// TwinCAT 3 PLC project WC1
// ProgramVersion: 3.1.4024.0
// libraries:
//   CmpBitmapPool, * (System)
//   Tc2_ModbusSrv, * (Beckhoff Automation GmbH)
//   Tc2_Standard, * (Beckhoff Automation GmbH)
//   Tc2_System, * (Beckhoff Automation GmbH)
//   Tc2_Utilities, * (Beckhoff Automation GmbH)
//   Tc3_Module, * (Beckhoff Automation GmbH)
//   VisuDialogs, * (System)
//   VisuSymbols,3.5.10.0,System
// project tree:
//   DUTs/ SEQ_NAME.TcDUT
//   / GlobalTextList.TcGTLO, PlcTask.TcTTO, Visualization Manager.TcVMO (not stored), VISU_TASK.TcTTO
//   POUs/Auto_Seq/ AUTO_MODE.TcPOU, FB_RunLayerPad.TcPOU, IF_RACK_CHECK.TcPOU, SEQ_A1.TcPOU, SEQ_A2.TcPOU, SEQ_A3.TcPOU, SEQ_A4.TcPOU, SEQ_A5.TcPOU, SEQ_B1.TcPOU, SEQ_B2.TcPOU, SEQ_B3.TcPOU, SEQ_B4.TcPOU, SEQ_B5.TcPOU, SEQ_COSMO.TcPOU, SEQ_CR_PICK.TcPOU, SEQ_CR_PLACE.TcPOU, SEQ_FG.TcPOU, SEQ_FG_A.TcPOU, SEQ_LYR_PD0.TcPOU, SEQ_RW.TcPOU
//   POUs/ COOL_RACK.TcPOU, ESTOP.TcPOU, INFEED_RACK.TcPOU, JIG.TcPOU, LOGGING.TcPOU, MAIN.TcPOU, RESET_SEQ.TcPOU, LOG_TIME_STAMP.TcPOU, SAFETY_SENSOR.TcPOU, TL.TcPOU, TORCHCLEAN.TcPOU, User.TcTLO
//   POUs/GVLs/ GVL.TcGVL, MSG.TcGVL
//   POUs/Kuka IO/ KR1.TcPOU, KR2.TcPOU, KR3.TcPOU, KR4.TcPOU, KR5.TcPOU, KUKA_IO.TcPOU
//   POUs/LOGGING/ FB_UpdateTimeStamp.TcPOU, LOGFILE.TcPOU, LOGPROCESS.TcPOU
//   VISUs/Dialog/ MSG_BOX_RESET.TcVIS, MSG_EOAT.TcVIS, MSG_EOAT_SUCTION.TcVIS, MSG_KR2_BP.TcVIS, MSG_KR4_BP.TcVIS, MSG_KR1_BP.TcVIS, MSG_KR3_BP.TcVIS
//   VISUs/ Footer_Main.TcVIS, Footer_Back.TcVIS, Header.TcVIS, ImagePool.TcIPO (not stored), PAGE_InfeedRack.TcVIS, PAGE_COSMO.TcVIS, PAGE_JIG_C.TcVIS, PAGE_CoolRack.TcVIS, PAGE_JIG_A.TcVIS, PAGE_JIG_B.TcVIS, PAGE_KR1_Tab.TcVIS, PAGE_KR1_Tab_1_100.TcVIS, PAGE_KR1_Tab_1_200.TcVIS, PAGE_MAIN_1.TcVIS, PAGE_TTorch.TcVIS, PAGE_MAIN.TcVIS, PAGE_KR2.TcVIS, PAGE_KR3.TcVIS, PAGE_KR4.TcVIS, PAGE_KR5.TcVIS, PAGE_KR1.TcVIS
// real-time tasks:
//   TASK PlcTask: cycle T#10ms, priority 6, ADS port 350
//   TASK VISU_TASK: cycle T#100000us, priority 8, ADS port 351
// I/O:
//   DEVICE Device 3 (EtherCAT), AmsNetId 169.254.168.184.4.1
//     Term 5 (EK1100) [EK1100 EtherCAT Coupler (2A E-Bus)]
//       Term 12 (EL1889) [EL1889 16Ch. Dig. Input 24V, 3ms, negative]
//       Term 13 (EL1889) [EL1889 16Ch. Dig. Input 24V, 3ms, negative]
//       Term 14 (EL2889) [EL2889 16Ch. Dig. Output 24V, 0.5A, negative]
//       Term 15 (EL9410) [EL9410 E-Bus Power Supplier  (Diagnostics)]
//       Term 16 (EL6695) KR1(KR5) [EL6695 EtherCAT Bridge terminal (Primary)]
//       Term 17 (EL6695) KR2(KR3) [EL6695 EtherCAT Bridge terminal (Primary)]
//       Term 18 (EL6695) KR3(KR2) [EL6695 EtherCAT Bridge terminal (Primary)]
//       Term 19 (EL6695) KR4 [EL6695 EtherCAT Bridge terminal (Primary)]
//       Term 20 (EL6695) KR5(KR1) [EL6695 EtherCAT Bridge terminal (Primary)]
//       Term 21 (EL9011) [EL9011 End Terminal]
// variable links:
//   WC1/WC1 Instance <-> Device 3 (EtherCAT)/Term 5 (EK1100)/Term 12 (EL1889)
//     PlcTask Inputs/GVL.COSMO_NOTOK <-> Channel 12/COSMO NOTOK
//     PlcTask Inputs/GVL.COSMO_OK <-> Channel 11/COSMO OK
//     PlcTask Inputs/GVL.COSMO_Ready <-> Channel 10/COSMO READY
//     PlcTask Inputs/GVL.Conveyor_Full <-> Channel 14/CONVY FULL
//     PlcTask Inputs/GVL.JIGA_Ready <-> Channel 3/JIG A READY
//     PlcTask Inputs/GVL.JIGA_Standby <-> Channel 2/JIG A STANDBY
//     PlcTask Inputs/GVL.JIGB_Ready <-> Channel 5/JIG B READY
//     PlcTask Inputs/GVL.JIGB_Standby <-> Channel 4/JIG B STANDBY
//     PlcTask Inputs/GVL.JIGC_Ready <-> Channel 7/JIG C READY
//     PlcTask Inputs/GVL.JIGC_Standby <-> Channel 6/JIG C STANDBY
//     PlcTask Inputs/GVL.Rework_Empty <-> Channel 15/REWORK EMPTY
//     PlcTask Inputs/GVL.TTorch_Complete <-> Channel 9/TT COMPLETE
//     PlcTask Inputs/GVL.TTorch_Standy <-> Channel 8/TT STANDBY
//     PlcTask Inputs/GVL.VibBowl_Ready <-> Channel 13/VB READY
//     PlcTask Inputs/MAIN.btnEstop <-> Channel 1/Estop
//   WC1/WC1 Instance <-> Device 3 (EtherCAT)/Term 5 (EK1100)/Term 13 (EL1889)
//     PlcTask Inputs/GVL.JIGA_Complete <-> Channel 9/JIGA_Complete
//     PlcTask Inputs/GVL.JIGB_Complete <-> Channel 10/JIGB_Complete
//     PlcTask Inputs/GVL.JIGC_Complete <-> Channel 11/JIGC_Complete
//     PlcTask Inputs/MAIN.btnReset <-> Channel 3/RESET BTN
//     PlcTask Inputs/MAIN.btnStart <-> Channel 1/START BTN
//     PlcTask Inputs/MAIN.btnStop <-> Channel 2/STOP BTN
//     PlcTask Inputs/SAFETY_SENSOR.SENSOR_AIR_PRESSURE_HIGH <-> Channel 5/AirPressure_High
//     PlcTask Inputs/SAFETY_SENSOR.SENSOR_AIR_PRESSURE_OK <-> Channel 4/GasPressure_OK
//     PlcTask Inputs/SAFETY_SENSOR.SENSOR_GAS_PRESSURE_HIGH <-> Channel 7/GasPressure_High
//     PlcTask Inputs/SAFETY_SENSOR.SENSOR_GAS_PRESSURE_OK <-> Channel 6/GasPressure_OK
//     PlcTask Inputs/SAFETY_SENSOR.SENSOR_SAFETY_DOOR_CLOSE <-> Channel 8/SafetyDoor
//   WC1/WC1 Instance <-> Device 3 (EtherCAT)/Term 5 (EK1100)/Term 14 (EL2889)
//     PlcTask Outputs/GVL.COSMO_Run <-> Channel 8/COSMO RUN
//     PlcTask Outputs/GVL.JIGA_Clamp <-> Channel 1/JIG A CLAMP
//     PlcTask Outputs/GVL.JIGA_Release <-> Channel 2/JIG A RELEASE
//     PlcTask Outputs/GVL.JIGB_Clamp <-> Channel 3/JIG B CLAMP
//     PlcTask Outputs/GVL.JIGB_Release <-> Channel 4/JIG B RELEASE
//     PlcTask Outputs/GVL.JIGC_Clamp <-> Channel 5/JIG C CLAMP
//     PlcTask Outputs/GVL.JIGC_Release <-> Channel 6/JIG C RELEASE
//     PlcTask Outputs/GVL.TTorch_Run <-> Channel 7/TT RUN
//     PlcTask Outputs/TL.TL_Buzzer <-> Channel 12/TL BUZZER
//     PlcTask Outputs/TL.TL_Ember <-> Channel 10/TL EMBER
//     PlcTask Outputs/TL.TL_Green <-> Channel 9/TL GREEN
//     PlcTask Outputs/TL.TL_Red <-> Channel 11/TL RED
//   WC1/WC1 Instance <-> Device 3 (EtherCAT)/Term 5 (EK1100)/Term 16 (EL6695) KR1(KR5)
//     PlcTask Inputs/KR1.PLC_I_AXIS[{1..6}] <-> IO Inputs/Var {229..234}  (6 links)
//     PlcTask Inputs/KR1.PLC_I_CURR[{1..6}] <-> IO Inputs/Var {235..240}  (6 links)
//     PlcTask Inputs/KR1.PLC_I_PROG{1..8} <-> IO Inputs/Var {220..227}  (8 links)
//     PlcTask Inputs/KR1.PLC_I_SYS <-> IO Inputs/Var 228
//     PlcTask Inputs/KR1.PLC_I_TEMP[{1..6}] <-> IO Inputs/Var {241..246}  (6 links)
//     PlcTask Outputs/KR1.PLC_O_PROG{1..8} <-> IO Outputs/Var {247..254}  (8 links)
//     PlcTask Outputs/KR1.PLC_O_SYS <-> IO Outputs/Var 255
//   WC1/WC1 Instance <-> Device 3 (EtherCAT)/Term 5 (EK1100)/Term 17 (EL6695) KR2(KR3)
//     PlcTask Inputs/KR2.PLC_I_AXIS[1] <-> IO Inputs/Var 51
//     PlcTask Inputs/KR2.PLC_I_AXIS[2] <-> IO Inputs/Var 134
//     PlcTask Inputs/KR2.PLC_I_AXIS[3] <-> IO Inputs/Var 135
//     PlcTask Inputs/KR2.PLC_I_AXIS[4] <-> IO Inputs/Var 136
//     PlcTask Inputs/KR2.PLC_I_AXIS[5] <-> IO Inputs/Var 137
//     PlcTask Inputs/KR2.PLC_I_AXIS[6] <-> IO Inputs/Var 138
//     PlcTask Inputs/KR2.PLC_I_CURR[{1..6}] <-> IO Inputs/Var {179..184}  (6 links)
//     PlcTask Inputs/KR2.PLC_I_PROG1 <-> IO Inputs/Var 47
//     PlcTask Inputs/KR2.PLC_I_PROG2 <-> IO Inputs/Var 48
//     PlcTask Inputs/KR2.PLC_I_SYS <-> IO Inputs/Var 50
//     PlcTask Inputs/KR2.PLC_I_TEMP[1] <-> IO Inputs/Var 185
//     PlcTask Inputs/KR2.PLC_I_TEMP[2] <-> IO Inputs/Var 186
//     PlcTask Inputs/KR2.PLC_I_TEMP[3] <-> IO Inputs/Var 187
//     PlcTask Inputs/KR2.PLC_I_TEMP[4] <-> IO Inputs/Var 188
//     PlcTask Inputs/KR2.PLC_I_TEMP[5] <-> IO Inputs/Var 189
//     PlcTask Inputs/KR2.PLC_I_TEMP[6] <-> IO Inputs/Var 196
//     PlcTask Outputs/KR2.PLC_O_PROG1 <-> IO Outputs/Var 190
//     PlcTask Outputs/KR2.PLC_O_PROG2 <-> IO Outputs/Var 191
//     PlcTask Outputs/KR2.PLC_O_SYS <-> IO Outputs/Var 192
//   WC1/WC1 Instance <-> Device 3 (EtherCAT)/Term 5 (EK1100)/Term 18 (EL6695) KR3(KR2)
//     PlcTask Inputs/KR3.PLC_I_AXIS[1] <-> IO Inputs/Var 46
//     PlcTask Inputs/KR3.PLC_I_AXIS[2] <-> IO Inputs/Var 47
//     PlcTask Inputs/KR3.PLC_I_AXIS[3] <-> IO Inputs/Var 48
//     PlcTask Inputs/KR3.PLC_I_AXIS[4] <-> IO Inputs/Var 49
//     PlcTask Inputs/KR3.PLC_I_AXIS[5] <-> IO Inputs/Var 114
//     PlcTask Inputs/KR3.PLC_I_AXIS[6] <-> IO Inputs/Var 115
//     PlcTask Inputs/KR3.PLC_I_CURR[1] <-> IO Inputs/Var 116
//     PlcTask Inputs/KR3.PLC_I_CURR[2] <-> IO Inputs/Var 117
//     PlcTask Inputs/KR3.PLC_I_CURR[3] <-> IO Inputs/Var 118
//     PlcTask Inputs/KR3.PLC_I_CURR[4] <-> IO Inputs/Var 119
//     PlcTask Inputs/KR3.PLC_I_CURR[5] <-> IO Inputs/Var 197
//     PlcTask Inputs/KR3.PLC_I_CURR[6] <-> IO Inputs/Var 198
//     PlcTask Inputs/KR3.PLC_I_PROG1 <-> IO Inputs/Var 44
//     PlcTask Inputs/KR3.PLC_I_SYS <-> IO Inputs/Var 45
//     PlcTask Inputs/KR3.PLC_I_TEMP[{1..6}] <-> IO Inputs/Var {199..204}  (6 links)
//     PlcTask Outputs/KR3.PLC_O_PROG1 <-> IO Outputs/Var 205
//     PlcTask Outputs/KR3.PLC_O_SYS <-> IO Outputs/Var 206
//   WC1/WC1 Instance <-> Device 3 (EtherCAT)/Term 5 (EK1100)/Term 19 (EL6695) KR4
//     PlcTask Inputs/KR4.PLC_I_AXIS[{1..6}] <-> IO Inputs/Var {234..239}  (6 links)
//     PlcTask Inputs/KR4.PLC_I_CURR[{1..6}] <-> IO Inputs/Var {240..245}  (6 links)
//     PlcTask Inputs/KR4.PLC_I_PROG1 <-> IO Inputs/Var 232
//     PlcTask Inputs/KR4.PLC_I_SYS <-> IO Inputs/Var 233
//     PlcTask Inputs/KR4.PLC_I_TEMP[{1..6}] <-> IO Inputs/Var {246..251}  (6 links)
//     PlcTask Outputs/KR4.PLC_O_PROG1 <-> IO Outputs/Var 252
//     PlcTask Outputs/KR4.PLC_O_SYS <-> IO Outputs/Var 253
//   WC1/WC1 Instance <-> Device 3 (EtherCAT)/Term 5 (EK1100)/Term 20 (EL6695) KR5(KR1)
//     PlcTask Inputs/KR5.PLC_I_AXIS[1] <-> IO Inputs/Var 7
//     PlcTask Inputs/KR5.PLC_I_AXIS[2] <-> IO Inputs/Var 8
//     PlcTask Inputs/KR5.PLC_I_AXIS[3] <-> IO Inputs/Var 9
//     PlcTask Inputs/KR5.PLC_I_AXIS[4] <-> IO Inputs/Var 10
//     PlcTask Inputs/KR5.PLC_I_AXIS[5] <-> IO Inputs/Var 75
//     PlcTask Inputs/KR5.PLC_I_AXIS[6] <-> IO Inputs/Var 76
//     PlcTask Inputs/KR5.PLC_I_CURR[1] <-> IO Inputs/Var 77
//     PlcTask Inputs/KR5.PLC_I_CURR[2] <-> IO Inputs/Var 78
//     PlcTask Inputs/KR5.PLC_I_CURR[3] <-> IO Inputs/Var 79
//     PlcTask Inputs/KR5.PLC_I_CURR[4] <-> IO Inputs/Var 80
//     PlcTask Inputs/KR5.PLC_I_CURR[5] <-> IO Inputs/Var 298
//     PlcTask Inputs/KR5.PLC_I_CURR[6] <-> IO Inputs/Var 299
//     PlcTask Inputs/KR5.PLC_I_PROG1 <-> IO Inputs/Var 5
//     PlcTask Inputs/KR5.PLC_I_SYS <-> IO Inputs/Var 6
//     PlcTask Inputs/KR5.PLC_I_TEMP[{1..6}] <-> IO Inputs/Var {300..305}  (6 links)
//     PlcTask Outputs/KR5.PLC_O_PROG1 <-> IO Outputs/Var 306
//     PlcTask Outputs/KR5.PLC_O_SYS <-> IO Outputs/Var 307

CONFIGURATION WC1
    RESOURCE PLC ON TwinCAT3
        TASK PlcTask(INTERVAL := T#10ms, PRIORITY := 6);
        TASK VISU_TASK(INTERVAL := T#100000us, PRIORITY := 8);
        PROGRAM MAIN WITH PlcTask : MAIN;
        PROGRAM VisuElems_Visu_Prg WITH VISU_TASK : VisuElems.Visu_Prg;
    END_RESOURCE
END_CONFIGURATION

// ---- DUTs/SEQ_NAME.TcDUT
{attribute 'qualified_only'}
{attribute 'strict'}
TYPE SEQ_NAME :
(
	INITIATE,
	IFRACK_PICK,
	PLACE_TO_JIG_A,
	JIG_A_CLAMP,
	JIG_A_WELDING,
	JIG_A_TO_JIG_B,
	JIG_B_CLAMP,
	JIG_B_WELDING,
	JIG_B_TO_TT,
	TT_WELDING,
	TT_WELD_COMPLETE,
	TT_TO_JIG_C,
	BRACKET_TO_JIG_C,
	JIG_C_CLAMP,
	JIG_C_WELDING,
	JIG_C_PICK,
	PLACE_TO_CR,
	END
);
END_TYPE

// ---- POUs/GVLs/GVL.TcGVL
{attribute 'qualified_only'}

VAR_GLOBAL PERSISTENT
	iCooling_Time 	: INT :=30;
	
	CRTimer			: ARRAY [1..21] OF INT;
	CR_NextPickNum	: UINT;
	CR_NextPlaceNum	: UINT;
	
	monthly_output	: USINT;
	weekly_output	: USINT;
	daily_output	: USINT;
	
	Basket_A_Counter : UINT;
	Basket_B_Counter : UINT;
	
	Fail_Counter	: USINT;
	Pass_Counter	: USINT;
	Rework_Counter	: USINT;	
	
	KR1_EOAT_FILL	: BOOL;
	KR1_EOAT_SUCTION: BOOL;
	
	ClearError		: BOOL;
		
	LAYERPAD0	: BOOL := FALSE;
END_VAR

VAR_GLOBAL
	//IO -> JIG
	JIGA_Standby 	AT %I*	: BOOL;
	JIGA_Ready	 	AT %I*	: BOOL;
	JIGA_Complete 	AT %I*	: BOOL;
	JIGB_Standby 	AT %I*	: BOOL;
	JIGB_Ready	 	AT %I*	: BOOL;
	JIGB_Complete 	AT %I*	: BOOL;
	JIGC_Standby 	AT %I*	: BOOL;
	JIGC_Ready 		AT %I*	: BOOL;
	JIGC_Complete 	AT %I*	: BOOL;
	JIGA_Clamp 	 	AT %Q*	: BOOL;
	JIGA_Release 	AT %Q*	: BOOL;
	JIGB_Clamp 		AT %Q*	: BOOL;
	JIGB_Release	AT %Q*	: BOOL;
	JIGC_Clamp 		AT %Q*	: BOOL;
	JIGC_Release 	AT %Q*	: BOOL;
	
	//IO -> TWIN TORCH
	TTorch_Standy   AT %I*	: BOOL;
	TTorch_Complete AT %I*	: BOOL;
	TTorch_Run	 	AT %Q*	: BOOL;
	
	//IO -> VIBRATOR BOWL
	VibBowl_Ready	AT %I*	: BOOL;
	
	//IO -> CONVEYOR & REWORK JIG
	Conveyor_Full	AT %I*	: BOOL;
	Rework_Empty	AT %I*	: BOOL;
	
	//IO -> COSMO
	COSMO_OK	 	AT %I*	: BOOL;
	COSMO_NOTOK	 	AT %I*	: BOOL;
	COSMO_Ready	 	AT %I*	: BOOL;
	COSMO_Run	 	AT %Q*	: BOOL;
	
	//Variable
	JIG_ERROR	: BOOL := FALSE;
	
	//Kuka
	KR2_bypass	: BOOL := FALSE;
	KR5_bypass	: BOOL := FALSE;
	KR4_bypass	: BOOL := FALSE;
	KR3_bypass	: BOOL := FALSE;
	KR1_bypass	: BOOL := FALSE;
	
	//pack
	LAYERPAD	: BOOL := FALSE;
	COSMO_UNLOAD: BOOL := FALSE;
	
END_VAR

// ---- POUs/GVLs/MSG.TcGVL
{attribute 'qualified_only'}
VAR_GLOBAL
	EVENT_BTN			: STRING := '[BTN] ';
	EVENT_PAGE			: STRING := '[PAGE] ';
	EVENT_PROCESS		: STRING := '[PROCESS] ';
	
	COMP_A5				: STRING := '|A5| ';
	COMP_A4				: STRING := '|A4| ';
	COMP_A3				: STRING := '|A3| ';
	COMP_A2				: STRING := '|A2| ';
	COMP_A1				: STRING := '|A1| ';
	COMP_B5				: STRING := '|B5| ';
	COMP_B4				: STRING := '|B4| ';
	COMP_B3				: STRING := '|B3| ';
	COMP_B2				: STRING := '|B2| ';
	COMP_B1				: STRING := '|B1| ';
	COMP_TT				: STRING := '|T.T| ';
	COMP_IR				: STRING := '|I.R| ';
	COMP_CR				: STRING := '|C.R| ';
	COMP_CM				: STRING := '|C.M| ';
	COMP_RW				: STRING := '|R.W| ';
	COMP_FG				: STRING := '|F.G| ';
	COMP_KR1			: STRING := '|KR1| ';
	COMP_KR2			: STRING := '|KR2| ';
	COMP_KR3			: STRING := '|KR3| ';
	COMP_KR4			: STRING := '|KR4| ';
	COMP_KR5			: STRING := '|KR5| ';
	COMP_JIGA			: STRING := '|JigA| ';
	COMP_JIGB			: STRING := '|JigB| ';
	COMP_JIGC			: STRING := '|JigC| ';
	COMP_HMI			: STRING := '|HMI| ';
	COMP_OP_BTN			: STRING := '|OP_BTN| ';
	
// STATUS MSG ---------------------------------------------------------		
	STATUS_RUN			: STRING := ' (RUN)';
	STATUS_ACK			: STRING := ' (ACK)';
	STATUS_DONE			: STRING := ' (DONE)';
	STATUS_COMP			: STRING := ' (COMPLETE)';
	STATUS_ERROR		: STRING := ' (ERROR)';
	STATUS_END			: STRING := ' (END)';

// ACTION MSG ---------------------------------------------------------	
	ACTION_ESTOP			: STRING := 'Emergency Stop';
	ACTION_START			: STRING := 'Start Production';
	ACTION_STOP		  		: STRING := 'Stop Production';
	ACTION_RESET			: STRING := 'Reset Production';
	ACTION_CLEAR_ERROR		: STRING := 'Clear Error';
	
	ACTION_RESET_KUKA		: STRING := 'Reset Kuka';
	ACTION_NEXTSTEP			: STRING := 'Next Step';
	ACTION_LOGIN			: STRING := 'User Login';
	ACTION_LOGOUT			: STRING := 'User Logout';
	ACTION_BSKTA_PLUS		: STRING := 'Basket A +';
	ACTION_BSKTA_MINUS		: STRING := 'Basket A -';
	ACTION_BSKTB_PLUS		: STRING := 'Basket B +';
	ACTION_BSKTB_MINUS		: STRING := 'Basket B -';
	ACTION_BACK				: STRING := 'Back';
	ACTION_KR1				: STRING := 'KR1';
	ACTION_KR2				: STRING := 'KR2';
	ACTION_KR3				: STRING := 'KR3';
	ACTION_KR4				: STRING := 'KR4';
	ACTION_KR5				: STRING := 'KR5';
	ACTION_COSMO			: STRING := 'Cosmo';
	ACTION_COSMO_PLACE		: STRING := 'Cosmo Place';
	ACTION_COOLRACK			: STRING := 'Cooling Rack';
	ACTION_INFEEDRACK		: STRING := 'Infeed Rack';
	ACTION_INFEEDRACK_PICK 	: STRING := 'Infeed Rack Pick';
	ACTION_TT				: STRING := 'TwinTorch';
	ACTION_JIGA				: STRING := 'Jig A';
	ACTION_JIGB				: STRING := 'Jig B';
	ACTION_JIGC				: STRING := 'Jig C';
	ACTION_TORCHCLEAN		: STRING := 'Torch Clean' ;
	ACTION_EOAT_YES			: STRING := 'Magnet Flag On';
	ACTION_EOAT_NO			: STRING := 'Magnet Flag Off';
	ACTION_SET_TIME			: STRING := 'Set Cooling Time';
	
	ACTION_MOVE_ENABLE		: STRING := 'Move Enable';
	ACTION_DRIVE_OFF		: STRING := 'Drive Off';
	ACTION_IO_ACT			: STRING := 'IO Act';
	ACTION_EXT_START		: STRING := 'Ext Start';
	ACTION_CONF_MESS		: STRING := 'Conf Mess';
	ACTION_DRIVE_ON			: STRING := 'Drive On';
	ACTION_PGNO_FBIT		: STRING := 'PGNO Fbit';
	ACTION_PGNO_VALID		: STRING := 'PGNO Valid';
	ACTION_PGNO_PARITY		: STRING := 'PGNO Parity';
	ACTION_1032				: STRING := '1032';
	ACTION_1036				: STRING := '1036';
	ACTION_1037				: STRING := '1037';
	ACTION_1038				: STRING := '1038';
	ACTION_1039				: STRING := '1039';
	ACTION_1040				: STRING := '1040';
	ACTION_1041				: STRING := '1041';
	ACTION_1042				: STRING := '1042';
	
	ACTION_200				: STRING := '200';
	ACTION_201				: STRING := '201';
	ACTION_202				: STRING := '202';
	ACTION_203				: STRING := '203';
	ACTION_204				: STRING := '204';
	ACTION_205				: STRING := '205';
	ACTION_206				: STRING := '206';
	ACTION_207				: STRING := '207';
	ACTION_208				: STRING := '208';
	ACTION_209				: STRING := '209';
	ACTION_210				: STRING := '210';
	ACTION_211				: STRING := '211';
	ACTION_212				: STRING := '212';
	ACTION_213				: STRING := '213';
	ACTION_214				: STRING := '214';
	ACTION_215				: STRING := '215';
	ACTION_216				: STRING := '216';
	ACTION_217				: STRING := '217';
	ACTION_218				: STRING := '218';
	ACTION_219				: STRING := '219';
	ACTION_220				: STRING := '220';
	ACTION_221				: STRING := '221';
	ACTION_222				: STRING := '222';
	ACTION_223				: STRING := '223';
	ACTION_224				: STRING := '224';
	ACTION_225				: STRING := '225';
	ACTION_226				: STRING := '226';
	ACTION_227				: STRING := '227';
	ACTION_228				: STRING := '228';
	ACTION_229				: STRING := '229';
	ACTION_230				: STRING := '230';
	ACTION_231				: STRING := '231';
	ACTION_300				: STRING := '300';
	ACTION_301				: STRING := '301';
	ACTION_302				: STRING := '302';
	ACTION_303				: STRING := '303';
	ACTION_304				: STRING := '304';
	ACTION_305				: STRING := '305';
	ACTION_306				: STRING := '306';
	ACTION_307				: STRING := '307';
	
	ACTION_GET_MAGNET		: STRING := 'Get Magnet';
	ACTION_REMOVE_MAGNET	: STRING := 'Remove Magnet';
	ACTION_GET_SUCTION		: STRING := 'Get Suction';
	ACTION_REMOVE_SUCTION	: STRING := 'Remove Suction';
	ACTION_GO_HOME			: STRING := 'Go Home';
	ACTION_COSMO_TO_PITSTOP	: STRING := 'Cosmo to Pitstop';
	ACTION_COSMO_TO_CNVYR	: STRING := 'Cosmo to Conveyor';
	ACTION_COSMO_PASS		: STRING := 'Cosmo Pass';
	ACTION_COSMO_FAIL		: STRING := 'Cosmo Fail';
	ACTION_REWORK_IN		: STRING := 'Rework In';
	ACTION_GET_LAYER_PAD	: STRING := 'Get Layer Pad';
	ACTION_PLACE_LAYER_PAD	: STRING := 'Place Layer Pad';
	ACTION_FGA_POS1			: STRING := 'FG Basket A POS 1';
	ACTION_FGA_POS2			: STRING := 'FG Basket A POS 2';
	ACTION_FGA_POS3			: STRING := 'FG Basket A POS 3';
	ACTION_FGA_POS4			: STRING := 'FG Basket A POS 4';
	ACTION_FGA_POS5			: STRING := 'FG Basket A POS 5';
	ACTION_FGA_POS6			: STRING := 'FG Basket A POS 6';
	ACTION_FGA_POS7			: STRING := 'FG Basket A POS 7';
	ACTION_FGA_POS8			: STRING := 'FG Basket A POS 8';
	ACTION_FGA_POS9			: STRING := 'FG Basket A POS 9';
	ACTION_FGA_POS10		: STRING := 'FG Basket A POS 10';
	ACTION_FGA_POS11		: STRING := 'FG Basket A POS 11';
	ACTION_FGA_POS12		: STRING := 'FG Basket A POS 12';
	ACTION_FGA_POS13		: STRING := 'FG Basket A POS 13';
	ACTION_FGA_POS14		: STRING := 'FG Basket A POS 14';
	ACTION_FGA_POS15		: STRING := 'FG Basket A POS 15';
	ACTION_FGA_POS16		: STRING := 'FG Basket A POS 16';
	ACTION_FGA_POS17		: STRING := 'FG Basket A POS 17';
	ACTION_FGA_POS18		: STRING := 'FG Basket A POS 18';
	ACTION_FGA_POS19		: STRING := 'FG Basket A POS 19';
	ACTION_FGA_POS20		: STRING := 'FG Basket A POS 20';
	ACTION_FGA_POS21		: STRING := 'FG Basket A POS 21';
	ACTION_FGA_POS22		: STRING := 'FG Basket A POS 22';
	ACTION_FGA_POS23		: STRING := 'FG Basket A POS 23';
	ACTION_FGA_POS24		: STRING := 'FG Basket A POS 24';
	ACTION_FGA_POS25		: STRING := 'FG Basket A POS 25';
	ACTION_FGA_POS26		: STRING := 'FG Basket A POS 26';
	ACTION_FGA_POS27		: STRING := 'FG Basket A POS 27';
	ACTION_FGA_POS28		: STRING := 'FG Basket A POS 28';
	ACTION_FGA_POS29		: STRING := 'FG Basket A POS 29';
	ACTION_FGA_POS30		: STRING := 'FG Basket A POS 30';
	ACTION_FGA_POS31		: STRING := 'FG Basket A POS 31';
	ACTION_FGA_POS32		: STRING := 'FG Basket A POS 32';
	ACTION_FGA_POS33		: STRING := 'FG Basket A POS 33';
	ACTION_FGA_POS34		: STRING := 'FG Basket A POS 34';
	ACTION_FGA_POS35		: STRING := 'FG Basket A POS 35';
	ACTION_FGA_POS36		: STRING := 'FG Basket A POS 36';
	ACTION_FGA_POS37		: STRING := 'FG Basket A POS 37';
	ACTION_FGA_POS38		: STRING := 'FG Basket A POS 38';
	ACTION_FGA_POS39		: STRING := 'FG Basket A POS 39';
	ACTION_FGA_POS40		: STRING := 'FG Basket A POS 40';
	ACTION_FGA_POS41		: STRING := 'FG Basket A POS 41';
	ACTION_FGA_POS42		: STRING := 'FG Basket A POS 42';
	ACTION_FGA_POS43		: STRING := 'FG Basket A POS 43';
	ACTION_FGA_POS44		: STRING := 'FG Basket A POS 44';
	ACTION_FGA_POS45		: STRING := 'FG Basket A POS 45';
	ACTION_FGA_POS46		: STRING := 'FG Basket A POS 46';
	ACTION_FGA_POS47		: STRING := 'FG Basket A POS 47';
	ACTION_FGA_POS48		: STRING := 'FG Basket A POS 48';
	ACTION_FGA_POS49		: STRING := 'FG Basket A POS 49';
	ACTION_FGA_POS50		: STRING := 'FG Basket A POS 50';
	ACTION_FGA_POS51		: STRING := 'FG Basket A POS 51';
	ACTION_FGA_POS52		: STRING := 'FG Basket A POS 52';
	ACTION_FGA_POS53		: STRING := 'FG Basket A POS 53';
	ACTION_FGA_POS54		: STRING := 'FG Basket A POS 54';
	ACTION_FGA_POS55		: STRING := 'FG Basket A POS 55';
	ACTION_FGA_POS56		: STRING := 'FG Basket A POS 56';
	ACTION_FGA_POS57		: STRING := 'FG Basket A POS 57';
	ACTION_FGA_POS58		: STRING := 'FG Basket A POS 58';
	ACTION_FGA_POS59		: STRING := 'FG Basket A POS 59';
	ACTION_FGA_POS60		: STRING := 'FG Basket A POS 60';
	ACTION_FGA_POS61		: STRING := 'FG Basket A POS 61';
	ACTION_FGA_POS62		: STRING := 'FG Basket A POS 62';
	ACTION_FGA_POS63		: STRING := 'FG Basket A POS 63';
	ACTION_FGA_POS64		: STRING := 'FG Basket A POS 64';
	ACTION_FGA_POS65		: STRING := 'FG Basket A POS 65';
	ACTION_FGA_POS66		: STRING := 'FG Basket A POS 66';
	ACTION_FGA_POS67		: STRING := 'FG Basket A POS 67';
	ACTION_FGA_POS68		: STRING := 'FG Basket A POS 68';
	ACTION_FGA_POS69		: STRING := 'FG Basket A POS 69';
	ACTION_FGA_POS70		: STRING := 'FG Basket A POS 70';
	ACTION_FGA_POS71		: STRING := 'FG Basket A POS 71';
	ACTION_FGA_POS72		: STRING := 'FG Basket A POS 72';
	ACTION_FGA_POS73		: STRING := 'FG Basket A POS 73';
	ACTION_FGA_POS74		: STRING := 'FG Basket A POS 74';
	ACTION_FGA_POS75		: STRING := 'FG Basket A POS 75';
	ACTION_FGA_POS76		: STRING := 'FG Basket A POS 76';
	ACTION_FGA_POS77		: STRING := 'FG Basket A POS 77';
	ACTION_FGA_POS78		: STRING := 'FG Basket A POS 78';
	ACTION_FGA_POS79		: STRING := 'FG Basket A POS 79';
	ACTION_FGA_POS80		: STRING := 'FG Basket A POS 80';
	ACTION_FGA_POS81		: STRING := 'FG Basket A POS 81';
	ACTION_FGA_POS82		: STRING := 'FG Basket A POS 82';
	ACTION_FGA_POS83		: STRING := 'FG Basket A POS 83';
	ACTION_FGA_POS84		: STRING := 'FG Basket A POS 84';
	ACTION_FGA_POS85		: STRING := 'FG Basket A POS 85';
	ACTION_FGA_POS86		: STRING := 'FG Basket A POS 86';
	ACTION_FGA_POS87		: STRING := 'FG Basket A POS 87';
	ACTION_FGA_POS88		: STRING := 'FG Basket A POS 88';
	ACTION_FGA_POS89		: STRING := 'FG Basket A POS 89';
	ACTION_FGA_POS90		: STRING := 'FG Basket A POS 90';
	ACTION_FGA_POS91		: STRING := 'FG Basket A POS 91';
	ACTION_FGA_POS92		: STRING := 'FG Basket A POS 92';
	ACTION_FGA_POS93		: STRING := 'FG Basket A POS 93';
	ACTION_FGA_POS94		: STRING := 'FG Basket A POS 94';
	ACTION_FGA_POS95		: STRING := 'FG Basket A POS 95';
	ACTION_FGA_POS96		: STRING := 'FG Basket A POS 96';
	ACTION_FGA_POS97		: STRING := 'FG Basket A POS 97';
	ACTION_FGA_POS98		: STRING := 'FG Basket A POS 98';
	ACTION_FGA_POS99		: STRING := 'FG Basket A POS 99';
	ACTION_FGA_POS100		: STRING := 'FG Basket A POS 100';
	ACTION_FGA_POS101		: STRING := 'FG Basket A POS 101';
	ACTION_FGA_POS102		: STRING := 'FG Basket A POS 102';
	ACTION_FGA_POS103		: STRING := 'FG Basket A POS 103';
	ACTION_FGA_POS104		: STRING := 'FG Basket A POS 104';
	ACTION_FGA_POS105		: STRING := 'FG Basket A POS 105';
	ACTION_FGA_POS106		: STRING := 'FG Basket A POS 106';
	ACTION_FGA_POS107		: STRING := 'FG Basket A POS 107';
	ACTION_FGA_POS108		: STRING := 'FG Basket A POS 108';
	ACTION_FGA_POS109		: STRING := 'FG Basket A POS 109';
	ACTION_FGA_POS110		: STRING := 'FG Basket A POS 110';
	ACTION_FGA_POS111		: STRING := 'FG Basket A POS 111';
	ACTION_FGA_POS112		: STRING := 'FG Basket A POS 112';
	ACTION_FGA_POS113		: STRING := 'FG Basket A POS 113';
	ACTION_FGA_POS114		: STRING := 'FG Basket A POS 114';
	ACTION_FGA_POS115		: STRING := 'FG Basket A POS 115';
	ACTION_FGA_POS116		: STRING := 'FG Basket A POS 116';
	ACTION_FGA_POS117		: STRING := 'FG Basket A POS 117';
	ACTION_FGA_POS118		: STRING := 'FG Basket A POS 118';
	ACTION_FGA_POS119		: STRING := 'FG Basket A POS 119';
	ACTION_FGA_POS120		: STRING := 'FG Basket A POS 120';
	ACTION_FGA_POS121		: STRING := 'FG Basket A POS 121';
	ACTION_FGA_POS122		: STRING := 'FG Basket A POS 122';
	ACTION_FGA_POS123		: STRING := 'FG Basket A POS 123';
	ACTION_FGA_POS124		: STRING := 'FG Basket A POS 124';
	ACTION_FGA_POS125		: STRING := 'FG Basket A POS 125';
	ACTION_FGA_POS126		: STRING := 'FG Basket A POS 126';
	ACTION_FGA_POS127		: STRING := 'FG Basket A POS 127';
	ACTION_FGA_POS128		: STRING := 'FG Basket A POS 128';
	ACTION_FGA_POS129		: STRING := 'FG Basket A POS 129';
	ACTION_FGA_POS130		: STRING := 'FG Basket A POS 130';
	ACTION_FGA_POS131		: STRING := 'FG Basket A POS 131';
	ACTION_FGA_POS132		: STRING := 'FG Basket A POS 132';
	ACTION_FGA_POS133		: STRING := 'FG Basket A POS 133';
	ACTION_FGA_POS134		: STRING := 'FG Basket A POS 134';
	ACTION_FGA_POS135		: STRING := 'FG Basket A POS 135';
	ACTION_FGA_POS136		: STRING := 'FG Basket A POS 136';
	ACTION_FGA_POS137		: STRING := 'FG Basket A POS 137';
	ACTION_FGA_POS138		: STRING := 'FG Basket A POS 138';
	ACTION_FGA_POS139		: STRING := 'FG Basket A POS 139';
	ACTION_FGA_POS140		: STRING := 'FG Basket A POS 140';
	ACTION_FGA_POS141		: STRING := 'FG Basket A POS 141';
	ACTION_FGA_POS142		: STRING := 'FG Basket A POS 142';
	ACTION_FGA_POS143		: STRING := 'FG Basket A POS 143';
	ACTION_FGA_POS144		: STRING := 'FG Basket A POS 144';
	ACTION_FGA_POS145		: STRING := 'FG Basket A POS 145';
	ACTION_FGA_POS146		: STRING := 'FG Basket A POS 146';
	ACTION_FGA_POS147		: STRING := 'FG Basket A POS 147';
	ACTION_FGA_POS148		: STRING := 'FG Basket A POS 148';
	ACTION_FGA_POS149		: STRING := 'FG Basket A POS 149';
	ACTION_FGA_POS150		: STRING := 'FG Basket A POS 150';
	ACTION_FGA_POS151		: STRING := 'FG Basket A POS 151';
	ACTION_FGA_POS152		: STRING := 'FG Basket A POS 152';
	ACTION_FGA_POS153		: STRING := 'FG Basket A POS 153';
	ACTION_FGA_POS154		: STRING := 'FG Basket A POS 154';
	ACTION_FGA_POS155		: STRING := 'FG Basket A POS 155';
	ACTION_FGA_POS156		: STRING := 'FG Basket A POS 156';
	ACTION_FGA_POS157		: STRING := 'FG Basket A POS 157';
	ACTION_FGA_POS158		: STRING := 'FG Basket A POS 158';
	ACTION_FGA_POS159		: STRING := 'FG Basket A POS 159';
	ACTION_FGA_POS160		: STRING := 'FG Basket A POS 160';
	ACTION_FGA_POS161		: STRING := 'FG Basket A POS 161';
	ACTION_FGA_POS162		: STRING := 'FG Basket A POS 162';
	ACTION_FGA_POS163		: STRING := 'FG Basket A POS 163';
	ACTION_FGA_POS164		: STRING := 'FG Basket A POS 164';
	ACTION_FGA_POS165		: STRING := 'FG Basket A POS 165';
	ACTION_FGA_POS166		: STRING := 'FG Basket A POS 166';
	ACTION_FGA_POS167		: STRING := 'FG Basket A POS 167';
	ACTION_FGA_POS168		: STRING := 'FG Basket A POS 168';
	ACTION_FGA_POS169		: STRING := 'FG Basket A POS 169';
	ACTION_FGA_POS170		: STRING := 'FG Basket A POS 170';
	ACTION_FGA_POS171		: STRING := 'FG Basket A POS 171';
	ACTION_FGA_POS172		: STRING := 'FG Basket A POS 172';
	ACTION_FGA_POS173		: STRING := 'FG Basket A POS 173';
	ACTION_FGA_POS174		: STRING := 'FG Basket A POS 174';
	ACTION_FGA_POS175		: STRING := 'FG Basket A POS 175';
	ACTION_FGA_POS176		: STRING := 'FG Basket A POS 176';
	ACTION_FGA_POS177		: STRING := 'FG Basket A POS 177';
	ACTION_FGA_POS178		: STRING := 'FG Basket A POS 178';
	ACTION_FGA_POS179		: STRING := 'FG Basket A POS 179';
	ACTION_FGA_POS180		: STRING := 'FG Basket A POS 180';
	ACTION_FGA_POS181		: STRING := 'FG Basket A POS 181';
	ACTION_FGA_POS182		: STRING := 'FG Basket A POS 182';
	ACTION_FGA_POS183		: STRING := 'FG Basket A POS 183';
	ACTION_FGA_POS184		: STRING := 'FG Basket A POS 184';
	ACTION_FGA_POS185		: STRING := 'FG Basket A POS 185';
	ACTION_FGA_POS186		: STRING := 'FG Basket A POS 186';
	ACTION_FGA_POS187		: STRING := 'FG Basket A POS 187';
	ACTION_FGA_POS188		: STRING := 'FG Basket A POS 188';
	ACTION_FGA_POS189		: STRING := 'FG Basket A POS 189';
	ACTION_FGA_POS190		: STRING := 'FG Basket A POS 190';
	ACTION_FGA_POS191		: STRING := 'FG Basket A POS 191';
	ACTION_FGA_POS192		: STRING := 'FG Basket A POS 192';
	ACTION_FGA_POS193		: STRING := 'FG Basket A POS 193';
	ACTION_FGA_POS194		: STRING := 'FG Basket A POS 194';
	ACTION_FGA_POS195		: STRING := 'FG Basket A POS 195';
	ACTION_FGA_POS196		: STRING := 'FG Basket A POS 196';
	ACTION_FGA_POS197		: STRING := 'FG Basket A POS 197';
	ACTION_FGA_POS198		: STRING := 'FG Basket A POS 198';
	ACTION_FGA_POS199		: STRING := 'FG Basket A POS 199';
	ACTION_FGA_POS200		: STRING := 'FG Basket A POS 200';
	ACTION_FGA_POS			: STRING := 'FG Basket A Pack';
	ACTION_FG_PACK			: STRING := 'FG Packing';
	ACTION_VB_TO_JIGC		: STRING := 'VB to JIG C';
	ACTION_JIGC_PICK		: STRING := 'JIG C Pick';
	ACTION_PLACE_TO_CR1		: STRING := 'Place to CR01';
	ACTION_PLACE_TO_CR2		: STRING := 'Place to CR02';
	ACTION_PLACE_TO_CR3		: STRING := 'Place to CR03';
	ACTION_PLACE_TO_CR4		: STRING := 'Place to CR04';
	ACTION_PLACE_TO_CR5		: STRING := 'Place to CR05';
	ACTION_PLACE_TO_CR6		: STRING := 'Place to CR06';
	ACTION_PLACE_TO_CR7		: STRING := 'Place to CR07';
	ACTION_PLACE_TO_CR8		: STRING := 'Place to CR08';
	ACTION_PLACE_TO_CR9		: STRING := 'Place to CR09';
	ACTION_PLACE_TO_CR10	: STRING := 'Place to CR10';
	ACTION_PLACE_TO_CR11	: STRING := 'Place to CR11';
	ACTION_PLACE_TO_CR12	: STRING := 'Place to CR12';
	ACTION_PLACE_TO_CR13	: STRING := 'Place to CR13';
	ACTION_PLACE_TO_CR14	: STRING := 'Place to CR14';
	ACTION_PLACE_TO_CR15	: STRING := 'Place to CR15';
	ACTION_PLACE_TO_CR16	: STRING := 'Place to CR16';
	ACTION_PLACE_TO_CR17	: STRING := 'Place to CR17';
	ACTION_PLACE_TO_CR18	: STRING := 'Place to CR18';
	ACTION_PLACE_TO_CR19	: STRING := 'Place to CR19';
	ACTION_PLACE_TO_CR20	: STRING := 'Place to CR20';
	ACTION_PLACE_TO_CR21	: STRING := 'Place to CR21';
	ACTION_PLACE_TO_CR		: STRING := 'Place to CR';
	ACTION_CR_TO_COSMO		: STRING := 'CR to COSMO';
	ACTION_CR_PICK			: STRING := 'CR Pick';
	ACTION_CR1_PICK			: STRING := 'CR01 Pick';
	ACTION_CR2_PICK			: STRING := 'CR02 Pick';
	ACTION_CR3_PICK			: STRING := 'CR03 Pick';
	ACTION_CR4_PICK			: STRING := 'CR04 Pick';
	ACTION_CR5_PICK			: STRING := 'CR05 Pick';
	ACTION_CR6_PICK			: STRING := 'CR06 Pick';
	ACTION_CR7_PICK			: STRING := 'CR07 Pick';
	ACTION_CR8_PICK			: STRING := 'CR08 Pick';
	ACTION_CR9_PICK			: STRING := 'CR09 Pick';
	ACTION_CR10_PICK		: STRING := 'CR10 Pick';
	ACTION_CR11_PICK		: STRING := 'CR11 Pick';
	ACTION_CR12_PICK		: STRING := 'CR12 Pick';
	ACTION_CR13_PICK		: STRING := 'CR13 Pick';
	ACTION_CR14_PICK		: STRING := 'CR14 Pick';
	ACTION_CR15_PICK		: STRING := 'CR15 Pick';
	ACTION_CR16_PICK		: STRING := 'CR16 Pick';
	ACTION_CR17_PICK		: STRING := 'CR17 Pick';
	ACTION_CR18_PICK		: STRING := 'CR18 Pick';
	ACTION_CR19_PICK		: STRING := 'CR19 Pick';
	ACTION_CR20_PICK		: STRING := 'CR20 Pick';
	ACTION_CR21_PICK		: STRING := 'CR21 Pick';
	ACTION_JIGA_WELDING		: STRING := 'JIG A Welding';
	ACTION_JIGB_WELDING		: STRING := 'JIG B Welding';
	ACTION_JIGC_WELDING		: STRING := 'JIG C Welding';
	ACTION_TORCH_CLEAN		: STRING := 'Torch Clean';	
	ACTION_JIGA_PLACE		: STRING := 'Place to JIG A';
	ACTION_JIGA_TO_JIGB		: STRING := 'JIG A to JIG B';
	ACTION_JIGB_TO_TT		: STRING := 'JIG B to TwinTorch';
	ACTION_TT_TO_JIGC		: STRING := 'TwinTorch to JIG C';
	ACTION_IF_A5			: STRING := 'Pick Infeed Rack A5';
	ACTION_IF_A4			: STRING := 'Pick Infeed Rack A4';
	ACTION_IF_A3			: STRING := 'Pick Infeed Rack A3';
	ACTION_IF_A2			: STRING := 'Pick Infeed Rack A2';
	ACTION_IF_A1			: STRING := 'Pick Infeed Rack A1';
	ACTION_IF_B5			: STRING := 'Pick Infeed Rack B5';
	ACTION_IF_B4			: STRING := 'Pick Infeed Rack B4';
	ACTION_IF_B3			: STRING := 'Pick Infeed Rack B3';
	ACTION_IF_B2			: STRING := 'Pick Infeed Rack B2';
	ACTION_IF_B1			: STRING := 'Pick Infeed Rack B1';
	ACTION_INIT				: STRING := 'Initiate';
	ACTION_JIGA_CLAMP		: STRING := 'JIG A Clamp';
	ACTION_JIGA_RELEASE		: STRING := 'JIG A Release';
	ACTION_JIGA_COMPLETE	: STRING := 'JIG A Complete';
	ACTION_JIGB_CLAMP		: STRING := 'JIG B Clamp';
	ACTION_JIGB_RELEASE		: STRING := 'JIG B Release';
	ACTION_JIGB_COMPLETE	: STRING := 'JIG B Complete';
	ACTION_JIGC_CLAMP		: STRING := 'JIG C Clamp';
	ACTION_JIGC_RELEASE		: STRING := 'JIG C Release';
	ACTION_JIGC_COMPLETE	: STRING := 'JIG C Complete';
	ACTION_TT_RUN			: STRING := 'TwinTorch Run';
	ACTION_IF_TO_CR			: STRING := 'Infeed Rack to Cooling Rack';
	ACTION_LYRPD_INIT		: STRING := 'Init Layer Pad';
END_VAR

// ---- POUs/MAIN.TcPOU
PROGRAM MAIN

VAR_INPUT
	btnEstop		AT %I* : BOOL;
	btnStart		AT %I* : BOOL;
	btnStop			AT %I* : BOOL;
	btnReset		AT %I* : BOOL;
	btn_Reset		: BOOL;
	btnSoftEstop	: BOOL;
	btnTorchClean	: BOOL;
	Kuka_Ready		: BOOL;
	LogText			: STRING;
	BTN_LOG			: BOOL;
	Reset_State	: BOOL;
END_VAR

VAR
	fb_TimeStamp	: FB_UpdateTimeStamp;
	ModbusOn	: TON;
	ModbusOff	: TON;
	bOn			: BOOL;
	bLastOn		: BOOL;
END_VAR

	// =============================== Estop
		IF NOT btnEStop OR btnSoftEstop THEN
			ESTOP(); 
		END_IF
		
	// =============================== Reset
		IF btn_Reset THEN
			Reset_State := TRUE; 
		END_IF	
		
		IF btnReset THEN
			Reset_State := TRUE;
			IF NOT Reset_State THEN
				LOGFILE( sLogEvent	 := MSG.EVENT_BTN,
						sLogComp	 := MSG.COMP_OP_BTN, 
						sLogAction	 := MSG.ACTION_RESET, 
						 logFlag	 := TRUE);
			END_IF
		END_IF
			
		IF Reset_State THEN
			RESET_SEQ();
		END_IF
		
	// =============================== Kuka Ready	
		IF KR1.KROnline AND KR2.KROnline AND KR3.KROnline AND KR4.KROnline AND KR5.KROnline THEN
				MAIN.Kuka_Ready := TRUE;
		ELSE
				MAIN.Kuka_Ready := FALSE;	
		END_IF
		
	// =============================== Programme	
	fb_TimeStamp();
	IF fb_TimeStamp.timeValid THEN
			KUKA_IO();
			INFEED_RACK();
			COOL_RACK();
			JIG();
			AUTO_MODE();
			SAFETY_SENSOR();
			TL();
			
			//======================================= Modbus
			//Off time
			ModbusOn(IN:= NOT ModbusOff.Q, PT:= T#1S, Q=> bOn , ET=> );
			//On time
			ModbusOff(IN:= bOn, PT:= T#1S, Q=> , ET=> );
				
			IF bOn <> bLastOn THEN
				IF bON THEN
					COOL_RACK.bstart_Read := INFEED_RACK.bstart_Read := TRUE;
				ELSE
					COOL_RACK.bstart_Read := INFEED_RACK.bstart_Read := FALSE;
				END_IF
			END_IF
			bLastOn := bOn;
			// ================================================
		
			// ======================================= Torch Clean
			IF btnTorchClean THEN 
				TORCHCLEAN(); 
			ELSE 
				TORCHCLEAN.process_A:=0; 
			END_IF
		
			// ======================================= Operator Button
			IF btnStart THEN
				IF NOT AUTO_MODE.AutoMode THEN
					AUTO_MODE.Halt_Production := FALSE;
					LOGFILE( sLogEvent	 := MSG.EVENT_BTN,
							 sLogComp	 := MSG.COMP_OP_BTN, 
							 sLogAction	 := MSG.ACTION_START, 
							 logFlag	 := TRUE);
					AUTO_MODE.AutoMode := TRUE; 
					AUTO_MODE.Start_time := MAIN.fb_TimeStamp.SystemTime;
				ELSE
					AUTO_MODE.Halt_Production := FALSE;
					AUTO_MODE.AutoMode := TRUE; 
				END_IF
			END_IF
			
			IF btnStop THEN
				IF NOT AUTO_MODE.Halt_Production THEN
					LOGFILE( sLogEvent	 := MSG.EVENT_BTN,
							 sLogComp	 := MSG.COMP_OP_BTN, 
							 sLogAction	 := MSG.ACTION_STOP, 
							 logFlag	 := TRUE);
					KR1.bOutBit[1,0]:= FALSE;
					KR2.bOutBit[1,0]:= FALSE;
					KR3.bOutBit[1,0]:= FALSE;
					KR4.bOutBit[1,0]:= FALSE;
					KR5.bOutBit[1,0]:= FALSE;
					AUTO_MODE.Halt_Production := TRUE;
					AUTO_MODE.AutoMode := FALSE;
					Reset_State := FALSE;
				ELSE
					KR1.bOutBit[1,0]:= FALSE;
					KR2.bOutBit[1,0]:= FALSE;
					KR3.bOutBit[1,0]:= FALSE;
					KR4.bOutBit[1,0]:= FALSE;
					KR5.bOutBit[1,0]:= FALSE;
					AUTO_MODE.Halt_Production := TRUE;
					AUTO_MODE.AutoMode := FALSE;
					Reset_State := FALSE;
				END_IF
			END_IF
	END_IF

END_PROGRAM

// ---- POUs/LOGGING/FB_UpdateTimeStamp.TcPOU
FUNCTION_BLOCK FB_UpdateTimeStamp
VAR_INPUT
END_VAR
VAR_OUTPUT
	FullSystemTime	: STRING;
	SystemDate		: STRING;
	SystemTime		: STRING;
	SystemHour		: STRING;
	timeValid		: bool;
END_VAR
VAR
	fb_LocalTime	 : FB_LocalSystemTime;
END_VAR

fb_LocalTime(
		sNetID:= , 
		bEnable:= TRUE , 
		dwCycle:= 1, 
		dwOpt:= , 
		tTimeout:= ,
		bValid=> timeValid, 
		systemTime=> , 
		tzID=> );
		
IF fb_localTime.bValid THEN
	FullSystemTime 	:= SYSTEMTIME_TO_STRING(fb_LocalTime.systemTime);
	
	SystemDate		:= WORD_TO_STRING(fb_LocalTime.systemTime.wYear);
	SystemDate		:= CONCAT(SystemDate, '.');
	SystemDate		:= CONCAT(SystemDate, WORD_TO_STRING(fb_LocalTime.systemTime.wMonth));
	SystemDate		:= CONCAT(SystemDate, '.');
	SystemDate		:= CONCAT(SystemDate, WORD_TO_STRING(fb_LocalTime.systemTime.wDay));
	
	SystemTime		:= WORD_TO_STRING(fb_LocalTime.systemTime.wHour);
	SystemTime		:= CONCAT(SystemTime, ':');
	SystemTime		:= CONCAT(SystemTime, WORD_TO_STRING(fb_LocalTime.systemTime.wMinute));
	SystemTime		:= CONCAT(SystemTime, ':');
	SystemTime		:= CONCAT(SystemTime, WORD_TO_STRING(fb_LocalTime.systemTime.wSecond));
	
	SystemHour		:= WORD_TO_STRING(fb_LocalTime.systemTime.wHour);
END_IF

END_FUNCTION_BLOCK

// ---- POUs/ESTOP.TcPOU
PROGRAM ESTOP
VAR
	Bit1,Bit2 	: INT;
	LogText		: STRING;
END_VAR

	
	FOR Bit1 := 1 TO 30 BY 1 DO
		FOR Bit2 := 0 TO 7 BY 1 DO
			KR1.bOutBit[Bit1,Bit2] := FALSE;
		END_FOR
	END_FOR
	FOR Bit1 := 1 TO 8 BY 1 DO
		FOR Bit2 := 0 TO 7 BY 1 DO
			KR2.bOutBit[Bit1,Bit2] := FALSE;
		END_FOR
	END_FOR
	FOR Bit1 := 1 TO 3 BY 1 DO
		FOR Bit2 := 0 TO 7 BY 1 DO
			KR3.bOutBit[Bit1,Bit2] := FALSE;
			KR4.bOutBit[Bit1,Bit2] := FALSE;
		END_FOR
	END_FOR
	FOR Bit1 := 1 TO 6 BY 1 DO
		FOR Bit2 := 0 TO 7 BY 1 DO
			KR5.bOutBit[Bit1,Bit2] := FALSE;
		END_FOR
	END_FOR

	RESET_SEQ.Reset_seq	:= 0;
	MAIN.btn_Reset	:= FALSE;
	Main.Reset_State := FALSE;
	AUTO_MODE.AutoMode := AUTO_MODE.next_step := FALSE;
	
	IF_RACK_CHECK.checkIn_A5 := IF_RACK_CHECK.checkIn_A4 := IF_RACK_CHECK.checkIn_A3 := IF_RACK_CHECK.checkIn_A2 := IF_RACK_CHECK.checkIn_A1 := 
	IF_RACK_CHECK.checkIn_B5 := IF_RACK_CHECK.checkIn_B4 := IF_RACK_CHECK.checkIn_B3 := IF_RACK_CHECK.checkIn_B2 := IF_RACK_CHECK.checkIn_B1 := FALSE;
	
	SEQ_A5.A5_sequence		:= SEQ_A4.A4_sequence		:= SEQ_A3.A3_sequence	:= SEQ_A2.A2_sequence	:= SEQ_A1.A1_sequence:=
	SEQ_B5.B5_sequence		:= SEQ_B4.B4_sequence		:= SEQ_B3.B3_sequence	:= SEQ_B2.B2_sequence	:= SEQ_B1.B1_sequence:=
	SEQ_CR_PICK.CR_sequence	:= SEQ_COSMO.COSMO_sequence	:= SEQ_RW.RW_sequence 	:= SEQ_FG.FG_sequence	:= 0;
	
	AUTO_MODE.IF_PICK		:= AUTO_MODE.JIGC_PICK		:= AUTO_MODE.CR_PICK		:=
	AUTO_MODE.JIGA_WELDING 	:= AUTO_MODE.JIGB_WELDING 	:= AUTO_MODE.JIGC_WELDING	:= AUTO_MODE.TT_WELDING   	:= 
	AUTO_MODE.JIGA_LOAD 	:= AUTO_MODE.JIGB_LOAD  	:= AUTO_MODE.JIGC_LOAD 		:= AUTO_MODE.TT_LOAD		:=
	GVL.JIGA_Clamp 			:= GVL.JIGB_Clamp 			:= GVL.JIGC_Clamp 			:= AUTO_MODE.CR_UNLOADING	:= 
	AUTO_MODE.COSMO_LOAD 	:= AUTO_MODE.COSMO_RUN 	 	:= AUTO_MODE.CLEAR_COSMO  	:= AUTO_MODE.KR1_PITSTOP 	:= 
	AUTO_MODE.FG_PACKING  	:= AUTO_MODE.RW_PACKING 	:= GVL.COSMO_Run			:= GVL.TTorch_Run 			:= FALSE;
	
	AUTO_MODE.JIGA_ErrorState := AUTO_MODE.JIGB_ErrorState := AUTO_MODE.JIGC_ErrorState := AUTO_MODE.TT_ErrorState := FALSE;

END_PROGRAM

// ---- POUs/Kuka IO/KR1.TcPOU
PROGRAM KR1
VAR_INPUT
	PLC_O_SYS 	AT %Q* : DWORD;
	PLC_O_PROG1 AT %Q* : DWORD;
	PLC_O_PROG2 AT %Q* : DWORD;
	PLC_O_PROG3 AT %Q* : DWORD;
	PLC_O_PROG4 AT %Q* : DWORD;
	PLC_O_PROG5 AT %Q* : DWORD;
	PLC_O_PROG6 AT %Q* : DWORD;
	PLC_O_PROG7 AT %Q* : DWORD;
	PLC_O_PROG8 AT %Q* : DWORD;
	
	PLC_I_SYS 	AT %I* : DWORD;
	PLC_I_PROG1 AT %I* : DWORD;
	PLC_I_PROG2 AT %I* : DWORD;
	PLC_I_PROG3 AT %I* : DWORD;
	PLC_I_PROG4 AT %I* : DWORD;
	PLC_I_PROG5 AT %I* : DWORD;
	PLC_I_PROG6 AT %I* : DWORD;
	PLC_I_PROG7 AT %I* : DWORD;
	PLC_I_PROG8 AT %I* : DWORD;
	PLC_I_AXIS 	AT %I* : ARRAY[1..6] OF DWORD;
	PLC_I_CURR	AT %I* : ARRAY[1..6] OF DWORD;
	PLC_I_TEMP	AT %I* : ARRAY[1..6] OF DWORD;
	
	KR1_Estop		: BOOL;
	Idle			: BOOL;
	NoMotion		: BOOL;
	KROnline		: BOOL;
	KR_ProgReady	: BOOL;
	
	bOutBit : ARRAY [1..30,0..7] OF BOOL;
	bInBit  : ARRAY [1..30,0..7] OF BOOL;
	
	index		: USINT;
	index1		: USINT;
	
	dAxis		: ARRAY[1..6] OF DWORD;
	dCurr		: ARRAY[1..6] OF DWORD;
	dTemp		: ARRAY[1..6] OF DWORD;
END_VAR


	//If Soft EStop is pressed, turn off 1027 ~ 1034
	IF KR1_Estop THEN		
		bOutBit[1,0]:=bOutBit[1,1]:=bOutBit[1,2]:=bOutBit[1,3]:=
		bOutBit[1,4]:=bOutBit[1,5]:=bOutBit[1,6]:=bOutBit[1,7]:=FALSE;
	END_IF

	//Idle 	
	IF 	PLC_I_PROG1 = 1 AND PLC_I_PROG2 = 1 AND PLC_I_PROG3 = 1 AND PLC_I_PROG4 = 1 AND 
		PLC_I_PROG5 = 1 AND PLC_I_PROG6 = 1 AND PLC_I_PROG7 = 1 AND PLC_I_PROG8 = 1 THEN 
			Idle := TRUE;
	ELSE
			Idle := FALSE;	
	END_IF
	
	//Online
	IF bInBit[1,0] OR bInBit[1,3] THEN
		KROnline := TRUE;
	ELSE
		KROnline := FALSE;
	END_IF

	//Program Ready
	IF bInBit[1,6] AND bInBit[2,4] THEN
		KR_ProgReady := TRUE;
	ELSE
		KR_ProgReady := FALSE;
	END_IF
	
	// ======================================================================== System IO
	// Data In
	FOR index := 0 TO 31 BY 1 DO
		IF index < 8 THEN
			bInBit[1,index] := DWORD_TO_BOOL( SHR(PLC_I_SYS,index) AND 1);
		ELSIF index > 7 AND index < 16 THEN
			bInBit[2,index-8] := DWORD_TO_BOOL( SHR(PLC_I_SYS,index) AND 1);
		END_IF
	END_FOR
	
	// Data Out
	PLC_O_SYS.0 := bOutBit[1,0]; // 1027 move_enable
	PLC_O_SYS.1 := bOutBit[1,1]; // 1028 Drive_off
	PLC_O_SYS.2 := bOutBit[1,2]; // 1029 IO_Activate
	PLC_O_SYS.3 := bOutBit[1,3]; // 1030 Ext_Start
	PLC_O_SYS.4 := bOutBit[1,4]; // 1031 Conf_mess
	PLC_O_SYS.5 := bOutBit[1,5]; // 1032 Drive_on
	PLC_O_SYS.6 := bOutBit[1,6]; // 1033 Pgno_Fbit
	PLC_O_SYS.7 := bOutBit[1,7]; // 1034 Pgno_Valid
	PLC_O_SYS.8 := bOutBit[2,0]; // 1035 Pgno_Parity
	
	// ===================================================================== Programme IO
	FOR index := 0 TO 31 BY 1 DO
		IF index < 8 THEN
			bInBit[3,index] := DWORD_TO_BOOL( SHR(PLC_I_PROG1,index) AND 1);
		ELSIF index > 7 AND index < 16 THEN
			bInBit[4,index-8] := DWORD_TO_BOOL( SHR(PLC_I_PROG1,index) AND 1);
		ELSIF index > 15 AND index < 24 THEN
			bInBit[5,index-16] := DWORD_TO_BOOL( SHR(PLC_I_PROG1,index) AND 1);
		ELSIF index > 23 THEN
			bInBit[6,index-24] := DWORD_TO_BOOL( SHR(PLC_I_PROG1,index) AND 1);
		END_IF
	END_FOR
	
	FOR index := 0 TO 31 BY 1 DO
		IF index < 8 THEN
			bInBit[7,index] := DWORD_TO_BOOL( SHR(PLC_I_PROG2,index) AND 1);
		ELSIF index > 7 AND index < 16 THEN
			bInBit[8,index-8] := DWORD_TO_BOOL( SHR(PLC_I_PROG2,index) AND 1);
		ELSIF index > 15 AND index < 24 THEN
			bInBit[9,index-16] := DWORD_TO_BOOL( SHR(PLC_I_PROG2,index) AND 1);
		ELSIF index > 23 THEN
			bInBit[10,index-24] := DWORD_TO_BOOL( SHR(PLC_I_PROG2,index) AND 1);
		END_IF
	END_FOR
	
	FOR index := 0 TO 31 BY 1 DO
		IF index < 8 THEN
			bInBit[11,index] := DWORD_TO_BOOL( SHR(PLC_I_PROG3,index) AND 1);
		ELSIF index > 7 AND index < 16 THEN
			bInBit[12,index-8] := DWORD_TO_BOOL( SHR(PLC_I_PROG3,index) AND 1);
		ELSIF index > 15 AND index < 24 THEN
			bInBit[13,index-16] := DWORD_TO_BOOL( SHR(PLC_I_PROG3,index) AND 1);
		ELSIF index > 23 THEN
			bInBit[14,index-24] := DWORD_TO_BOOL( SHR(PLC_I_PROG3,index) AND 1);
		END_IF
	END_FOR
	
	FOR index := 0 TO 31 BY 1 DO
		IF index < 8 THEN
			bInBit[15,index] := DWORD_TO_BOOL( SHR(PLC_I_PROG4,index) AND 1);
		ELSIF index > 7 AND index < 16 THEN
			bInBit[16,index-8] := DWORD_TO_BOOL( SHR(PLC_I_PROG4,index) AND 1);
		ELSIF index > 15 AND index < 24 THEN
			bInBit[17,index-16] := DWORD_TO_BOOL( SHR(PLC_I_PROG4,index) AND 1);
		ELSIF index > 23 THEN
			bInBit[18,index-24] := DWORD_TO_BOOL( SHR(PLC_I_PROG4,index) AND 1);
		END_IF
	END_FOR
	
	FOR index := 0 TO 31 BY 1 DO
		IF index < 8 THEN
			bInBit[19,index] := DWORD_TO_BOOL( SHR(PLC_I_PROG5,index) AND 1);
		ELSIF index > 7 AND index < 16 THEN
			bInBit[20,index-8] := DWORD_TO_BOOL( SHR(PLC_I_PROG5,index) AND 1);
		ELSIF index > 15 AND index < 24 THEN
			bInBit[21,index-16] := DWORD_TO_BOOL( SHR(PLC_I_PROG5,index) AND 1);
		ELSIF index > 23 THEN
			bInBit[22,index-24] := DWORD_TO_BOOL( SHR(PLC_I_PROG5,index) AND 1);
		END_IF
	END_FOR
	
	FOR index := 0 TO 31 BY 1 DO
		IF index < 8 THEN
			bInBit[23,index] := DWORD_TO_BOOL( SHR(PLC_I_PROG6,index) AND 1);
		ELSIF index > 7 AND index < 16 THEN
			bInBit[24,index-8] := DWORD_TO_BOOL( SHR(PLC_I_PROG6,index) AND 1);
		ELSIF index > 15 AND index < 24 THEN
			bInBit[25,index-16] := DWORD_TO_BOOL( SHR(PLC_I_PROG6,index) AND 1);
		ELSIF index > 23 THEN
			bInBit[26,index-24] := DWORD_TO_BOOL( SHR(PLC_I_PROG6,index) AND 1);
		END_IF
	END_FOR
	
	FOR index := 0 TO 31 BY 1 DO
		IF index < 8 THEN
			bInBit[27,index] := DWORD_TO_BOOL( SHR(PLC_I_PROG7,index) AND 1);
		ELSIF index > 7 AND index < 16 THEN
			bInBit[28,index-8] := DWORD_TO_BOOL( SHR(PLC_I_PROG7,index) AND 1);
		ELSIF index > 15 AND index < 24 THEN
			bInBit[29,index-16] := DWORD_TO_BOOL( SHR(PLC_I_PROG7,index) AND 1);
		ELSIF index > 23 THEN
			bInBit[30,index-24] := DWORD_TO_BOOL( SHR(PLC_I_PROG7,index) AND 1);
		END_IF
	END_FOR
	
	PLC_O_PROG1.0 := bOutBit[3,0]; // 200
	PLC_O_PROG1.1 := bOutBit[3,1]; // 201
	PLC_O_PROG1.2 := bOutBit[3,2]; // 202
	PLC_O_PROG1.3 := bOutBit[3,3]; // 203
	PLC_O_PROG1.4 := bOutBit[3,4]; // 204
	PLC_O_PROG1.5 := bOutBit[3,5]; // 205
	PLC_O_PROG1.6 := bOutBit[3,6]; // 206
	PLC_O_PROG1.7 := bOutBit[3,7]; // 207
	PLC_O_PROG1.8 := bOutBit[4,0]; // 208
	PLC_O_PROG1.9 := bOutBit[4,1]; // 209
	PLC_O_PROG1.10 := bOutBit[4,2]; // 210
	PLC_O_PROG1.11 := bOutBit[4,3]; // 211
	PLC_O_PROG1.12 := bOutBit[4,4]; // 212
	PLC_O_PROG1.13 := bOutBit[4,5]; // 213
	PLC_O_PROG1.14 := bOutBit[4,6]; // 214
	PLC_O_PROG1.15 := bOutBit[4,7]; // 215
	PLC_O_PROG1.16 := bOutBit[5,0]; // 216
	PLC_O_PROG1.17 := bOutBit[5,1]; // 217
	PLC_O_PROG1.18 := bOutBit[5,2]; // 218
	PLC_O_PROG1.19 := bOutBit[5,3]; // 219
	PLC_O_PROG1.20 := bOutBit[5,4]; // 220
	PLC_O_PROG1.21 := bOutBit[5,5]; // 221
	PLC_O_PROG1.22 := bOutBit[5,6]; // 222
	PLC_O_PROG1.23 := bOutBit[5,7]; // 223
	PLC_O_PROG1.24 := bOutBit[6,0]; // 224
	PLC_O_PROG1.25 := bOutBit[6,1]; // 225
	PLC_O_PROG1.26 := bOutBit[6,2]; // 226
	PLC_O_PROG1.27 := bOutBit[6,3]; // 227
	PLC_O_PROG1.28 := bOutBit[6,4]; // 228
	PLC_O_PROG1.29 := bOutBit[6,5]; // 229
	PLC_O_PROG1.30 := bOutBit[6,6]; // 230
	PLC_O_PROG1.31 := bOutBit[6,7]; // 231
	
	PLC_O_PROG2.0 := bOutBit[7,0]; // 232
	PLC_O_PROG2.1 := bOutBit[7,1]; // 233
	PLC_O_PROG2.2 := bOutBit[7,2]; // 234
	PLC_O_PROG2.3 := bOutBit[7,3]; // 235
	PLC_O_PROG2.4 := bOutBit[7,4]; // 236
	PLC_O_PROG2.5 := bOutBit[7,5]; // 237
	PLC_O_PROG2.6 := bOutBit[7,6]; // 238
	PLC_O_PROG2.7 := bOutBit[7,7]; // 239
	PLC_O_PROG2.8 := bOutBit[8,0]; // 240
	PLC_O_PROG2.9 := bOutBit[8,1]; // 241
	PLC_O_PROG2.10 := bOutBit[8,2]; // 242
	PLC_O_PROG2.11 := bOutBit[8,3]; // 243
	PLC_O_PROG2.12 := bOutBit[8,4]; // 244
	PLC_O_PROG2.13 := bOutBit[8,5]; // 245
	PLC_O_PROG2.14 := bOutBit[8,6]; // 246
	PLC_O_PROG2.15 := bOutBit[8,7]; // 247
	PLC_O_PROG2.16 := bOutBit[9,0]; // 248
	PLC_O_PROG2.17 := bOutBit[9,1]; // 249
	PLC_O_PROG2.18 := bOutBit[9,2]; // 250
	PLC_O_PROG2.19 := bOutBit[9,3]; // 251
	PLC_O_PROG2.20 := bOutBit[9,4]; // 252
	PLC_O_PROG2.21 := bOutBit[9,5]; // 253
	PLC_O_PROG2.22 := bOutBit[9,6]; // 254
	PLC_O_PROG2.23 := bOutBit[9,7]; // 255
	PLC_O_PROG2.24 := bOutBit[10,0]; // 256
	PLC_O_PROG2.25 := bOutBit[10,1]; // 257
	PLC_O_PROG2.26 := bOutBit[10,2]; // 258
	PLC_O_PROG2.27 := bOutBit[10,3]; // 259
	PLC_O_PROG2.28 := bOutBit[10,4]; // 260
	PLC_O_PROG2.29 := bOutBit[10,5]; // 261
	PLC_O_PROG2.30 := bOutBit[10,6]; // 262
	PLC_O_PROG2.31 := bOutBit[10,7]; // 263
	
	PLC_O_PROG3.0 := bOutBit[11,0]; // 264
	PLC_O_PROG3.1 := bOutBit[11,1]; // 265
	PLC_O_PROG3.2 := bOutBit[11,2]; // 266
	PLC_O_PROG3.3 := bOutBit[11,3]; // 267
	PLC_O_PROG3.4 := bOutBit[11,4]; // 268
	PLC_O_PROG3.5 := bOutBit[11,5]; // 269
	PLC_O_PROG3.6 := bOutBit[11,6]; // 270
	PLC_O_PROG3.7 := bOutBit[11,7]; // 271
	PLC_O_PROG3.8 := bOutBit[12,0]; // 272
	PLC_O_PROG3.9 := bOutBit[12,1]; // 273
	PLC_O_PROG3.10 := bOutBit[12,2]; // 274
	PLC_O_PROG3.11 := bOutBit[12,3]; // 275
	PLC_O_PROG3.12 := bOutBit[12,4]; // 276
	PLC_O_PROG3.13 := bOutBit[12,5]; // 277
	PLC_O_PROG3.14 := bOutBit[12,6]; // 278
	PLC_O_PROG3.15 := bOutBit[12,7]; // 279
	PLC_O_PROG3.16 := bOutBit[13,0]; // 280
	PLC_O_PROG3.17 := bOutBit[13,1]; // 281
	PLC_O_PROG3.18 := bOutBit[13,2]; // 282
	PLC_O_PROG3.19 := bOutBit[13,3]; // 283
	PLC_O_PROG3.20 := bOutBit[13,4]; // 284
	PLC_O_PROG3.21 := bOutBit[13,5]; // 285
	PLC_O_PROG3.22 := bOutBit[13,6]; // 286
	PLC_O_PROG3.23 := bOutBit[13,7]; // 287
	PLC_O_PROG3.24 := bOutBit[14,0]; // 288
	PLC_O_PROG3.25 := bOutBit[14,1]; // 289
	PLC_O_PROG3.26 := bOutBit[14,2]; // 290
	PLC_O_PROG3.27 := bOutBit[14,3]; // 291
	PLC_O_PROG3.28 := bOutBit[14,4]; // 292
	PLC_O_PROG3.29 := bOutBit[14,5]; // 293
	PLC_O_PROG3.30 := bOutBit[14,6]; // 294
	PLC_O_PROG3.31 := bOutBit[14,7]; // 295
	
	PLC_O_PROG4.0 := bOutBit[15,0]; // 296
	PLC_O_PROG4.1 := bOutBit[15,1]; // 297
	PLC_O_PROG4.2 := bOutBit[15,2]; // 298
	PLC_O_PROG4.3 := bOutBit[15,3]; // 299
	PLC_O_PROG4.4 := bOutBit[15,4]; // 300
	PLC_O_PROG4.5 := bOutBit[15,5]; // 301
	PLC_O_PROG4.6 := bOutBit[15,6]; // 302
	PLC_O_PROG4.7 := bOutBit[15,7]; // 303
	PLC_O_PROG4.8 := bOutBit[16,0]; // 304
	PLC_O_PROG4.9 := bOutBit[16,1]; // 305
	PLC_O_PROG4.10 := bOutBit[16,2]; // 306
	PLC_O_PROG4.11 := bOutBit[16,3]; // 307
	PLC_O_PROG4.12 := bOutBit[16,4]; // 308
	PLC_O_PROG4.13 := bOutBit[16,5]; // 309
	PLC_O_PROG4.14 := bOutBit[16,6]; // 310
	PLC_O_PROG4.15 := bOutBit[16,7]; // 311
	PLC_O_PROG4.16 := bOutBit[17,0]; // 312
	PLC_O_PROG4.17 := bOutBit[17,1]; // 313
	PLC_O_PROG4.18 := bOutBit[17,2]; // 314
	PLC_O_PROG4.19 := bOutBit[17,3]; // 315
	PLC_O_PROG4.20 := bOutBit[17,4]; // 316
	PLC_O_PROG4.21 := bOutBit[17,5]; // 317
	PLC_O_PROG4.22 := bOutBit[17,6]; // 318
	PLC_O_PROG4.23 := bOutBit[17,7]; // 319
	PLC_O_PROG4.24 := bOutBit[18,0]; // 320
	PLC_O_PROG4.25 := bOutBit[18,1]; // 321
	PLC_O_PROG4.26 := bOutBit[18,2]; // 322
	PLC_O_PROG4.27 := bOutBit[18,3]; // 323
	PLC_O_PROG4.28 := bOutBit[18,4]; // 324
	PLC_O_PROG4.29 := bOutBit[18,5]; // 325
	PLC_O_PROG4.30 := bOutBit[18,6]; // 326
	PLC_O_PROG4.31 := bOutBit[18,7]; // 327
	
	PLC_O_PROG5.0 := bOutBit[19,0]; // 328
	PLC_O_PROG5.1 := bOutBit[19,1]; // 329
	PLC_O_PROG5.2 := bOutBit[19,2]; // 330
	PLC_O_PROG5.3 := bOutBit[19,3]; // 331
	PLC_O_PROG5.4 := bOutBit[19,4]; // 332
	PLC_O_PROG5.5 := bOutBit[19,5]; // 333
	PLC_O_PROG5.6 := bOutBit[19,6]; // 334
	PLC_O_PROG5.7 := bOutBit[19,7]; // 335
	PLC_O_PROG5.8 := bOutBit[20,0]; // 336
	PLC_O_PROG5.9 := bOutBit[20,1]; // 337
	PLC_O_PROG5.10 := bOutBit[20,2]; // 338
	PLC_O_PROG5.11 := bOutBit[20,3]; // 339
	PLC_O_PROG5.12 := bOutBit[20,4]; // 340
	PLC_O_PROG5.13 := bOutBit[20,5]; // 341
	PLC_O_PROG5.14 := bOutBit[20,6]; // 342
	PLC_O_PROG5.15 := bOutBit[20,7]; // 343
	PLC_O_PROG5.16 := bOutBit[21,0]; // 344
	PLC_O_PROG5.17 := bOutBit[21,1]; // 345
	PLC_O_PROG5.18 := bOutBit[21,2]; // 346
	PLC_O_PROG5.19 := bOutBit[21,3]; // 347
	PLC_O_PROG5.20 := bOutBit[21,4]; // 348
	PLC_O_PROG5.21 := bOutBit[21,5]; // 349
	PLC_O_PROG5.22 := bOutBit[21,6]; // 350
	PLC_O_PROG5.23 := bOutBit[21,7]; // 351
	PLC_O_PROG5.24 := bOutBit[22,0]; // 352
	PLC_O_PROG5.25 := bOutBit[22,1]; // 353
	PLC_O_PROG5.26 := bOutBit[22,2]; // 354
	PLC_O_PROG5.27 := bOutBit[22,3]; // 355
	PLC_O_PROG5.28 := bOutBit[22,4]; // 356
	PLC_O_PROG5.29 := bOutBit[22,5]; // 357
	PLC_O_PROG5.30 := bOutBit[22,6]; // 358
	PLC_O_PROG5.31 := bOutBit[22,7]; // 359
	
	PLC_O_PROG6.0 := bOutBit[23,0]; // 360
	PLC_O_PROG6.1 := bOutBit[23,1]; // 361
	PLC_O_PROG6.2 := bOutBit[23,2]; // 362
	PLC_O_PROG6.3 := bOutBit[23,3]; // 363
	PLC_O_PROG6.4 := bOutBit[23,4]; // 364
	PLC_O_PROG6.5 := bOutBit[23,5]; // 365
	PLC_O_PROG6.6 := bOutBit[23,6]; // 366
	PLC_O_PROG6.7 := bOutBit[23,7]; // 367
	PLC_O_PROG6.8 := bOutBit[24,0]; // 368
	PLC_O_PROG6.9 := bOutBit[24,1]; // 369
	PLC_O_PROG6.10 := bOutBit[24,2]; // 370
	PLC_O_PROG6.11 := bOutBit[24,3]; // 371
	PLC_O_PROG6.12 := bOutBit[24,4]; // 372
	PLC_O_PROG6.13 := bOutBit[24,5]; // 373
	PLC_O_PROG6.14 := bOutBit[24,6]; // 374
	PLC_O_PROG6.15 := bOutBit[24,7]; // 375
	PLC_O_PROG6.16 := bOutBit[25,0]; // 376
	PLC_O_PROG6.17 := bOutBit[25,1]; // 377
	PLC_O_PROG6.18 := bOutBit[25,2]; // 378
	PLC_O_PROG6.19 := bOutBit[25,3]; // 379
	PLC_O_PROG6.20 := bOutBit[25,4]; // 380
	PLC_O_PROG6.21 := bOutBit[25,5]; // 381
	PLC_O_PROG6.22 := bOutBit[25,6]; // 382
	PLC_O_PROG6.23 := bOutBit[25,7]; // 383
	PLC_O_PROG6.24 := bOutBit[26,0]; // 384
	PLC_O_PROG6.25 := bOutBit[26,1]; // 385
	PLC_O_PROG6.26 := bOutBit[26,2]; // 386
	PLC_O_PROG6.27 := bOutBit[26,3]; // 387
	PLC_O_PROG6.28 := bOutBit[26,4]; // 388
	PLC_O_PROG6.29 := bOutBit[26,5]; // 389
	PLC_O_PROG6.30 := bOutBit[26,6]; // 390
	PLC_O_PROG6.31 := bOutBit[26,7]; // 391
	
	PLC_O_PROG7.0 := bOutBit[27,0]; // 392
	PLC_O_PROG7.1 := bOutBit[27,1]; // 393
	PLC_O_PROG7.2 := bOutBit[27,2]; // 394
	PLC_O_PROG7.3 := bOutBit[27,3]; // 395
	PLC_O_PROG7.4 := bOutBit[27,4]; // 396
	PLC_O_PROG7.5 := bOutBit[27,5]; // 397
	PLC_O_PROG7.6 := bOutBit[27,6]; // 398
	PLC_O_PROG7.7 := bOutBit[27,7]; // 399
	PLC_O_PROG7.8 := bOutBit[28,0]; // 400
	PLC_O_PROG7.9 := bOutBit[28,1]; // 401
	PLC_O_PROG7.10 := bOutBit[28,2]; // 402
	PLC_O_PROG7.11 := bOutBit[28,3]; // 403
	PLC_O_PROG7.12 := bOutBit[28,4]; // 404
	PLC_O_PROG7.13 := bOutBit[28,5]; // 405
	PLC_O_PROG7.14 := bOutBit[28,6]; // 406
	PLC_O_PROG7.15 := bOutBit[28,7]; // 407
	PLC_O_PROG7.16 := bOutBit[29,0]; // 408
	PLC_O_PROG7.17 := bOutBit[29,1]; // 409
	PLC_O_PROG7.18 := bOutBit[29,2]; // 410
	PLC_O_PROG7.19 := bOutBit[29,3]; // 411
	PLC_O_PROG7.20 := bOutBit[29,4]; // 412
	PLC_O_PROG7.21 := bOutBit[29,5]; // 413
	PLC_O_PROG7.22 := bOutBit[29,6]; // 414
	PLC_O_PROG7.23 := bOutBit[29,7]; // 415
	PLC_O_PROG7.24 := bOutBit[30,0]; // 416
	PLC_O_PROG7.25 := bOutBit[30,1]; // 417
	PLC_O_PROG7.26 := bOutBit[30,2]; // 418
	PLC_O_PROG7.27 := bOutBit[30,3]; // 419
	PLC_O_PROG7.28 := bOutBit[30,4]; // 420
	PLC_O_PROG7.29 := bOutBit[30,5]; // 421
	PLC_O_PROG7.30 := bOutBit[30,6]; // 422
	PLC_O_PROG7.31 := bOutBit[30,7]; // 423
	
	// ===================================================================== Robot Data
	FOR index1 := 1 TO 6 BY 1 DO
		FOR index := 0 TO 31 BY 1 DO
			dAxis[index1] := PLC_I_AXIS[index1];
			dCurr[index1] := PLC_I_CURR[index1];
			dTemp[index1] := PLC_I_TEMP[index1];
		END_FOR
	END_FOR
	
	
	
	
	
	
	
	
	
	
	
	
	
	
	
	
	
//	//================================ Function IO
	
//	PLC_O_D1.0 := bOutBit[1,0]; //1027 motion enable (on to start motor)
//	PLC_O_D1.1 := bOutBit[1,1]; //1028 Drives off (inverse) (on to start motor)
//	PLC_O_D1.2 := bOutBit[1,2]; //1029 Activate interface (on to start motor)
//	PLC_O_D1.3 := bOutBit[1,3]; //1030 Prog Start
//	PLC_O_D1.4 := bOutBit[1,4]; //1031 Acknowledge error msg
//	PLC_O_D1.5 := bOutBit[1,5]; //1032 Drives on
//	PLC_O_D1.6 := bOutBit[1,6]; //1033
//	PLC_O_D1.7 := bOutBit[1,7]; //1034
	
//	PLC_O_D2.0 := bOutBit[2,0]; //1035
//	PLC_O_D2.1 := bOutBit[2,1]; //1036
//	PLC_O_D2.2 := bOutBit[2,2]; //1037
//	PLC_O_D2.3 := bOutBit[2,3]; //1038
//	PLC_O_D2.4 := bOutBit[2,4]; //1039
//	PLC_O_D2.5 := bOutBit[2,5]; //1040
//	PLC_O_D2.6 := bOutBit[2,6]; //1041
//	PLC_O_D2.7 := bOutBit[2,7]; //1042
	
//	bInBit[1,0] := PLC_I_D1.0; //993
//	bInBit[1,1] := PLC_I_D1.1; //994
//	bInBit[1,2] := PLC_I_D1.2; //995
//	bInBit[1,3] := PLC_I_D1.3; //996
//	bInBit[1,4] := PLC_I_D1.4; //997
//	bInBit[1,5] := PLC_I_D1.5; //998
//	bInBit[1,6] := PLC_I_D1.6; //999
//	bInBit[1,7] := PLC_I_D1.7; //1000
	
//	bInBit[2,0] := PLC_I_D2.0; //1001
//	bInBit[2,1] := PLC_I_D2.1; //1002
//	bInBit[2,2] := PLC_I_D2.2; //1003
//	bInBit[2,3] := PLC_I_D2.3; //1004
//	bInBit[2,4] := PLC_I_D2.4; //1005
//	bInBit[2,5] := PLC_I_D2.5; //1006
//	bInBit[2,6] := PLC_I_D2.6; //1007
//	bInBit[2,7] := PLC_I_D2.7; //1008
	
//	//================================ Motion IO
	
//	IF NoMotion THEN
//		RETURN;
//	END_IF
	
//	PLC_O_D3.0 := bOutBit[3,0]; //200
//	PLC_O_D3.1 := bOutBit[3,1]; //201
//	PLC_O_D3.2 := bOutBit[3,2]; //202
//	PLC_O_D3.3 := bOutBit[3,3]; //203
//	PLC_O_D3.4 := bOutBit[3,4]; //204
//	PLC_O_D3.5 := bOutBit[3,5]; //205
//	PLC_O_D3.6 := bOutBit[3,6]; //206
//	PLC_O_D3.7 := bOutBit[3,7]; //207
	
//	PLC_O_D4.0 := bOutBit[4,0]; //208
//	PLC_O_D4.1 := bOutBit[4,1]; //209
//	PLC_O_D4.2 := bOutBit[4,2]; //210
//	PLC_O_D4.3 := bOutBit[4,3]; //211
//	PLC_O_D4.4 := bOutBit[4,4]; //212
//	PLC_O_D4.5 := bOutBit[4,5]; //213
//	PLC_O_D4.6 := bOutBit[4,6]; //214
//	PLC_O_D4.7 := bOutBit[4,7]; //215
	
//	PLC_O_D5.0 := bOutBit[5,0]; //216
//	PLC_O_D5.1 := bOutBit[5,1]; //217
//	PLC_O_D5.2 := bOutBit[5,2]; //218
//	PLC_O_D5.3 := bOutBit[5,3]; //219
//	PLC_O_D5.4 := bOutBit[5,4]; //220
//	PLC_O_D5.5 := bOutBit[5,5]; //221
//	PLC_O_D5.6 := bOutBit[5,6]; //222
//	PLC_O_D5.7 := bOutBit[5,7]; //223

//	PLC_O_D6.0 := bOutBit[6,0]; //224
//	PLC_O_D6.1 := bOutBit[6,1]; //225
//	PLC_O_D6.2 := bOutBit[6,2]; //226
//	PLC_O_D6.3 := bOutBit[6,3]; //227
//	PLC_O_D6.4 := bOutBit[6,4]; //228
//	PLC_O_D6.5 := bOutBit[6,5]; //229
//	PLC_O_D6.6 := bOutBit[6,6]; //230
//	PLC_O_D6.7 := bOutBit[6,7]; //231

//	PLC_O_D7.0 := bOutBit[7,0]; //224
//	PLC_O_D7.1 := bOutBit[7,1]; //225
//	PLC_O_D7.2 := bOutBit[7,2]; //227
//	PLC_O_D7.3 := bOutBit[7,3]; //227
//	PLC_O_D7.4 := bOutBit[7,4]; //228
//	PLC_O_D7.5 := bOutBit[7,5]; //229
//	PLC_O_D7.6 := bOutBit[7,6]; //230
//	PLC_O_D7.7 := bOutBit[7,7]; //231

//	PLC_O_D8.0 := bOutBit[8,0]; //224
//	PLC_O_D8.1 := bOutBit[8,1]; //225
//	PLC_O_D8.2 := bOutBit[8,2]; //228
//	PLC_O_D8.3 := bOutBit[8,3]; //227
//	PLC_O_D8.4 := bOutBit[8,4]; //228
//	PLC_O_D8.5 := bOutBit[8,5]; //229
//	PLC_O_D8.6 := bOutBit[8,6]; //230
//	PLC_O_D8.7 := bOutBit[8,7]; //231

//	PLC_O_D9.0 := bOutBit[9,0]; //224
//	PLC_O_D9.1 := bOutBit[9,1]; //225
//	PLC_O_D9.2 := bOutBit[9,2]; //226
//	PLC_O_D9.3 := bOutBit[9,3]; //227
//	PLC_O_D9.4 := bOutBit[9,4]; //228
//	PLC_O_D9.5 := bOutBit[9,5]; //229
//	PLC_O_D9.6 := bOutBit[9,6]; //230
//	PLC_O_D9.7 := bOutBit[9,7]; //231

//	PLC_O_D10.0 := bOutBit[10,0]; //224
//	PLC_O_D10.1 := bOutBit[10,1]; //225
//	PLC_O_D10.2 := bOutBit[10,2]; //226
//	PLC_O_D10.3 := bOutBit[10,3]; //227
//	PLC_O_D10.4 := bOutBit[10,4]; //228
//	PLC_O_D10.5 := bOutBit[10,5]; //229
//	PLC_O_D10.6 := bOutBit[10,6]; //230
//	PLC_O_D10.7 := bOutBit[10,7]; //231

//	PLC_O_D11.0 := bOutBit[11,0]; //224
//	PLC_O_D11.1 := bOutBit[11,1]; //225
//	PLC_O_D11.2 := bOutBit[11,2]; //226
//	PLC_O_D11.3 := bOutBit[11,3]; //227
//	PLC_O_D11.4 := bOutBit[11,4]; //228
//	PLC_O_D11.5 := bOutBit[11,5]; //229
//	PLC_O_D11.6 := bOutBit[11,6]; //230
//	PLC_O_D11.7 := bOutBit[11,7]; //231

//	PLC_O_D12.0 := bOutBit[12,0]; //224
//	PLC_O_D12.1 := bOutBit[12,1]; //225
//	PLC_O_D12.2 := bOutBit[12,2]; //226
//	PLC_O_D12.3 := bOutBit[12,3]; //227
//	PLC_O_D12.4 := bOutBit[12,4]; //228
//	PLC_O_D12.5 := bOutBit[12,5]; //229
//	PLC_O_D12.6 := bOutBit[12,6]; //230
//	PLC_O_D12.7 := bOutBit[12,7]; //231

//	PLC_O_D13.0 := bOutBit[13,0]; //224
//	PLC_O_D13.1 := bOutBit[13,1]; //225
//	PLC_O_D13.2 := bOutBit[13,2]; //226
//	PLC_O_D13.3 := bOutBit[13,3]; //227
//	PLC_O_D13.4 := bOutBit[13,4]; //228
//	PLC_O_D13.5 := bOutBit[13,5]; //229
//	PLC_O_D13.6 := bOutBit[13,6]; //230
//	PLC_O_D13.7 := bOutBit[13,7]; //231

//	PLC_O_D14.0 := bOutBit[14,0]; //224
//	PLC_O_D14.1 := bOutBit[14,1]; //225
//	PLC_O_D14.2 := bOutBit[14,2]; //226
//	PLC_O_D14.3 := bOutBit[14,3]; //227
//	PLC_O_D14.4 := bOutBit[14,4]; //228
//	PLC_O_D14.5 := bOutBit[14,5]; //229
//	PLC_O_D14.6 := bOutBit[14,6]; //230
//	PLC_O_D14.7 := bOutBit[14,7]; //231

//	PLC_O_D15.0 := bOutBit[15,0]; //224
//	PLC_O_D15.1 := bOutBit[15,1]; //225
//	PLC_O_D15.2 := bOutBit[15,2]; //226
//	PLC_O_D15.3 := bOutBit[15,3]; //227
//	PLC_O_D15.4 := bOutBit[15,4]; //228
//	PLC_O_D15.5 := bOutBit[15,5]; //229
//	PLC_O_D15.6 := bOutBit[15,6]; //230
//	PLC_O_D15.7 := bOutBit[15,7]; //231

//	PLC_O_D16.0 := bOutBit[16,0]; //224
//	PLC_O_D16.1 := bOutBit[16,1]; //225
//	PLC_O_D16.2 := bOutBit[16,2]; //226
//	PLC_O_D16.3 := bOutBit[16,3]; //227
//	PLC_O_D16.4 := bOutBit[16,4]; //228
//	PLC_O_D16.5 := bOutBit[16,5]; //229
//	PLC_O_D16.6 := bOutBit[16,6]; //230
//	PLC_O_D16.7 := bOutBit[16,7]; //231

//	PLC_O_D17.0 := bOutBit[17,0]; //224
//	PLC_O_D17.1 := bOutBit[17,1]; //225
//	PLC_O_D17.2 := bOutBit[17,2]; //226
//	PLC_O_D17.3 := bOutBit[17,3]; //227
//	PLC_O_D17.4 := bOutBit[17,4]; //228
//	PLC_O_D17.5 := bOutBit[17,5]; //229
//	PLC_O_D17.6 := bOutBit[17,6]; //230
//	PLC_O_D17.7 := bOutBit[17,7]; //231

//	PLC_O_D18.0 := bOutBit[18,0]; //224
//	PLC_O_D18.1 := bOutBit[18,1]; //225
//	PLC_O_D18.2 := bOutBit[18,2]; //226
//	PLC_O_D18.3 := bOutBit[18,3]; //227
//	PLC_O_D18.4 := bOutBit[18,4]; //228
//	PLC_O_D18.5 := bOutBit[18,5]; //229
//	PLC_O_D18.6 := bOutBit[18,6]; //230
//	PLC_O_D18.7 := bOutBit[18,7]; //231

//	PLC_O_D19.0 := bOutBit[19,0]; //224
//	PLC_O_D19.1 := bOutBit[19,1]; //225
//	PLC_O_D19.2 := bOutBit[19,2]; //226
//	PLC_O_D19.3 := bOutBit[19,3]; //227
//	PLC_O_D19.4 := bOutBit[19,4]; //228
//	PLC_O_D19.5 := bOutBit[19,5]; //229
//	PLC_O_D19.6 := bOutBit[19,6]; //230
//	PLC_O_D19.7 := bOutBit[19,7]; //231

//	PLC_O_D20.0 := bOutBit[20,0]; //224
//	PLC_O_D20.1 := bOutBit[20,1]; //225
//	PLC_O_D20.2 := bOutBit[20,2]; //226
//	PLC_O_D20.3 := bOutBit[20,3]; //227
//	PLC_O_D20.4 := bOutBit[20,4]; //228
//	PLC_O_D20.5 := bOutBit[20,5]; //229
//	PLC_O_D20.6 := bOutBit[20,6]; //230
//	PLC_O_D20.7 := bOutBit[20,7]; //231	

//	PLC_O_D21.0 := bOutBit[21,0]; //224
//	PLC_O_D21.1 := bOutBit[21,1]; //225
//	PLC_O_D21.2 := bOutBit[21,2]; //226
//	PLC_O_D21.3 := bOutBit[21,3]; //227
//	PLC_O_D21.4 := bOutBit[21,4]; //228
//	PLC_O_D21.5 := bOutBit[21,5]; //229
//	PLC_O_D21.6 := bOutBit[21,6]; //230
//	PLC_O_D21.7 := bOutBit[21,7]; //231

//	PLC_O_D22.0 := bOutBit[22,0]; //224
//	PLC_O_D22.1 := bOutBit[22,1]; //225
//	PLC_O_D22.2 := bOutBit[22,2]; //226
//	PLC_O_D22.3 := bOutBit[22,3]; //227
//	PLC_O_D22.4 := bOutBit[22,4]; //228
//	PLC_O_D22.5 := bOutBit[22,5]; //229
//	PLC_O_D22.6 := bOutBit[22,6]; //230
//	PLC_O_D22.7 := bOutBit[22,7]; //231

//	PLC_O_D23.0 := bOutBit[23,0]; //224
//	PLC_O_D23.1 := bOutBit[23,1]; //225
//	PLC_O_D23.2 := bOutBit[23,2]; //226
//	PLC_O_D23.3 := bOutBit[23,3]; //227
//	PLC_O_D23.4 := bOutBit[23,4]; //228
//	PLC_O_D23.5 := bOutBit[23,5]; //229
//	PLC_O_D23.6 := bOutBit[23,6]; //230
//	PLC_O_D23.7 := bOutBit[23,7]; //231

//	PLC_O_D24.0 := bOutBit[24,0]; //224
//	PLC_O_D24.1 := bOutBit[24,1]; //225
//	PLC_O_D24.2 := bOutBit[24,2]; //226
//	PLC_O_D24.3 := bOutBit[24,3]; //227
//	PLC_O_D24.4 := bOutBit[24,4]; //228
//	PLC_O_D24.5 := bOutBit[24,5]; //229
//	PLC_O_D24.6 := bOutBit[24,6]; //230
//	PLC_O_D24.7 := bOutBit[24,7]; //231

//	PLC_O_D25.0 := bOutBit[25,0]; //224
//	PLC_O_D25.1 := bOutBit[25,1]; //225
//	PLC_O_D25.2 := bOutBit[25,2]; //226
//	PLC_O_D25.3 := bOutBit[25,3]; //227
//	PLC_O_D25.4 := bOutBit[25,4]; //228
//	PLC_O_D25.5 := bOutBit[25,5]; //229
//	PLC_O_D25.6 := bOutBit[25,6]; //230
//	PLC_O_D25.7 := bOutBit[25,7]; //231

//	PLC_O_D26.0 := bOutBit[26,0]; //224
//	PLC_O_D26.1 := bOutBit[26,1]; //225
//	PLC_O_D26.2 := bOutBit[26,2]; //226
//	PLC_O_D26.3 := bOutBit[26,3]; //227
//	PLC_O_D26.4 := bOutBit[26,4]; //228
//	PLC_O_D26.5 := bOutBit[26,5]; //229
//	PLC_O_D26.6 := bOutBit[26,6]; //230
//	PLC_O_D26.7 := bOutBit[26,7]; //231

//	PLC_O_D27.0 := bOutBit[27,0]; //224
//	PLC_O_D27.1 := bOutBit[27,1]; //225
//	PLC_O_D27.2 := bOutBit[27,2]; //226
//	PLC_O_D27.3 := bOutBit[27,3]; //227
//	PLC_O_D27.4 := bOutBit[27,4]; //228
//	PLC_O_D27.5 := bOutBit[27,5]; //229
//	PLC_O_D27.6 := bOutBit[27,6]; //230
//	PLC_O_D27.7 := bOutBit[27,7]; //231

//	PLC_O_D28.0 := bOutBit[28,0]; //224
//	PLC_O_D28.1 := bOutBit[28,1]; //225
//	PLC_O_D28.2 := bOutBit[28,2]; //226
//	PLC_O_D28.3 := bOutBit[28,3]; //227
//	PLC_O_D28.4 := bOutBit[28,4]; //228
//	PLC_O_D28.5 := bOutBit[28,5]; //229
//	PLC_O_D28.6 := bOutBit[28,6]; //230
//	PLC_O_D28.7 := bOutBit[28,7]; //231

//	PLC_O_D29.0 := bOutBit[29,0]; //224
//	PLC_O_D29.1 := bOutBit[29,1]; //225
//	PLC_O_D29.2 := bOutBit[29,2]; //226
//	PLC_O_D29.3 := bOutBit[29,3]; //227
//	PLC_O_D29.4 := bOutBit[29,4]; //228
//	PLC_O_D29.5 := bOutBit[29,5]; //229
//	PLC_O_D29.6 := bOutBit[29,6]; //230
//	PLC_O_D29.7 := bOutBit[29,7]; //231

//	PLC_O_D30.0 := bOutBit[30,0]; //224
//	PLC_O_D30.1 := bOutBit[30,1]; //225
//	PLC_O_D30.2 := bOutBit[30,2]; //226
//	PLC_O_D30.3 := bOutBit[30,3]; //227
//	PLC_O_D30.4 := bOutBit[30,4]; //228
//	PLC_O_D30.5 := bOutBit[30,5]; //229
//	PLC_O_D30.6 := bOutBit[30,6]; //230
//	PLC_O_D30.7 := bOutBit[30,7]; //231

	
//	bInBit[3,0] := PLC_I_D3.0; //200
//	bInBit[3,1] := PLC_I_D3.1; //201
//	bInBit[3,2] := PLC_I_D3.2; //202
//	bInBit[3,3] := PLC_I_D3.3; //203
//	bInBit[3,4] := PLC_I_D3.4; //204
//	bInBit[3,5] := PLC_I_D3.5; //205
//	bInBit[3,6] := PLC_I_D3.6; //206
//	bInBit[3,7] := PLC_I_D3.7; //207
	
//	bInBit[4,0] := PLC_I_D4.0; //208
//	bInBit[4,1] := PLC_I_D4.1; //209
//	bInBit[4,2] := PLC_I_D4.2; //210
//	bInBit[4,3] := PLC_I_D4.3; //211
//	bInBit[4,4] := PLC_I_D4.4; //212
//	bInBit[4,5] := PLC_I_D4.5; //213
//	bInBit[4,6] := PLC_I_D4.6; //214
//	bInBit[4,7] := PLC_I_D4.7; //215
	
//	bInBit[5,0] := PLC_I_D5.0; //216
//	bInBit[5,1] := PLC_I_D5.1; //217
//	bInBit[5,2] := PLC_I_D5.2; //218
//	bInBit[5,3] := PLC_I_D5.3; //219
//	bInBit[5,4] := PLC_I_D5.4; //220
//	bInBit[5,5] := PLC_I_D5.5; //221
//	bInBit[5,6] := PLC_I_D5.6; //222
//	bInBit[5,7] := PLC_I_D5.7; //223
	
//	bInBit[6,0] := PLC_I_D6.0; //224
//	bInBit[6,1] := PLC_I_D6.1; //225
//	bInBit[6,2] := PLC_I_D6.2; //226
//	bInBit[6,3] := PLC_I_D6.3; //227
//	bInBit[6,4] := PLC_I_D6.4; //228
//	bInBit[6,5] := PLC_I_D6.5; //229
//	bInBit[6,6] := PLC_I_D6.6; //230
//	bInBit[6,7] := PLC_I_D6.7; //231
	
//	bInBit[7,0] := PLC_I_D7.0; //224
//	bInBit[7,1] := PLC_I_D7.1; //225
//	bInBit[7,2] := PLC_I_D7.2; //226
//	bInBit[7,3] := PLC_I_D7.3; //227
//	bInBit[7,4] := PLC_I_D7.4; //228
//	bInBit[7,5] := PLC_I_D7.5; //229
//	bInBit[7,6] := PLC_I_D7.6; //230
//	bInBit[7,7] := PLC_I_D7.7; //231
	
//	bInBit[8,0] := PLC_I_D8.0; //224
//	bInBit[8,1] := PLC_I_D8.1; //225
//	bInBit[8,2] := PLC_I_D8.2; //226
//	bInBit[8,3] := PLC_I_D8.3; //227
//	bInBit[8,4] := PLC_I_D8.4; //228
//	bInBit[8,5] := PLC_I_D8.5; //229
//	bInBit[8,6] := PLC_I_D8.6; //230
//	bInBit[8,7] := PLC_I_D8.7; //231
	
//	bInBit[9,0] := PLC_I_D9.0; //224
//	bInBit[9,1] := PLC_I_D9.1; //225
//	bInBit[9,2] := PLC_I_D9.2; //226
//	bInBit[9,3] := PLC_I_D9.3; //227
//	bInBit[9,4] := PLC_I_D9.4; //228
//	bInBit[9,5] := PLC_I_D9.5; //229
//	bInBit[9,6] := PLC_I_D9.6; //230
//	bInBit[9,7] := PLC_I_D9.7; //231
	
//	bInBit[10,0] := PLC_I_D10.0; //224
//	bInBit[10,1] := PLC_I_D10.1; //225
//	bInBit[10,2] := PLC_I_D10.2; //226
//	bInBit[10,3] := PLC_I_D10.3; //227
//	bInBit[10,4] := PLC_I_D10.4; //228
//	bInBit[10,5] := PLC_I_D10.5; //229
//	bInBit[10,6] := PLC_I_D10.6; //230
//	bInBit[10,7] := PLC_I_D10.7; //231
	
//	bInBit[11,0] := PLC_I_D11.0; //224
//	bInBit[11,1] := PLC_I_D11.1; //225
//	bInBit[11,2] := PLC_I_D11.2; //226
//	bInBit[11,3] := PLC_I_D11.3; //227
//	bInBit[11,4] := PLC_I_D11.4; //228
//	bInBit[11,5] := PLC_I_D11.5; //229
//	bInBit[11,6] := PLC_I_D11.6; //230
//	bInBit[11,7] := PLC_I_D11.7; //231
	
//	bInBit[12,0] := PLC_I_D12.0; //224
//	bInBit[12,1] := PLC_I_D12.1; //225
//	bInBit[12,2] := PLC_I_D12.2; //226
//	bInBit[12,3] := PLC_I_D12.3; //227
//	bInBit[12,4] := PLC_I_D12.4; //228
//	bInBit[12,5] := PLC_I_D12.5; //229
//	bInBit[12,6] := PLC_I_D12.6; //230
//	bInBit[12,7] := PLC_I_D12.7; //231
	
//	bInBit[13,0] := PLC_I_D13.0; //224
//	bInBit[13,1] := PLC_I_D13.1; //225
//	bInBit[13,2] := PLC_I_D13.2; //226
//	bInBit[13,3] := PLC_I_D13.3; //227
//	bInBit[13,4] := PLC_I_D13.4; //228
//	bInBit[13,5] := PLC_I_D13.5; //229
//	bInBit[13,6] := PLC_I_D13.6; //230
//	bInBit[13,7] := PLC_I_D13.7; //231
	
//	bInBit[14,0] := PLC_I_D14.0; //224
//	bInBit[14,1] := PLC_I_D14.1; //225
//	bInBit[14,2] := PLC_I_D14.2; //226
//	bInBit[14,3] := PLC_I_D14.3; //227
//	bInBit[14,4] := PLC_I_D14.4; //228
//	bInBit[14,5] := PLC_I_D14.5; //229
//	bInBit[14,6] := PLC_I_D14.6; //230
//	bInBit[14,7] := PLC_I_D14.7; //231
	
//	bInBit[15,0] := PLC_I_D15.0; //224
//	bInBit[15,1] := PLC_I_D15.1; //225
//	bInBit[15,2] := PLC_I_D15.2; //226
//	bInBit[15,3] := PLC_I_D15.3; //227
//	bInBit[15,4] := PLC_I_D15.4; //228
//	bInBit[15,5] := PLC_I_D15.5; //229
//	bInBit[15,6] := PLC_I_D15.6; //230
//	bInBit[15,7] := PLC_I_D15.7; //231
	
//	bInBit[16,0] := PLC_I_D16.0; //224
//	bInBit[16,1] := PLC_I_D16.1; //225
//	bInBit[16,2] := PLC_I_D16.2; //226
//	bInBit[16,3] := PLC_I_D16.3; //227
//	bInBit[16,4] := PLC_I_D16.4; //228
//	bInBit[16,5] := PLC_I_D16.5; //229
//	bInBit[16,6] := PLC_I_D16.6; //230
//	bInBit[16,7] := PLC_I_D16.7; //231
	
//	bInBit[17,0] := PLC_I_D17.0; //224
//	bInBit[17,1] := PLC_I_D17.1; //225
//	bInBit[17,2] := PLC_I_D17.2; //226
//	bInBit[17,3] := PLC_I_D17.3; //227
//	bInBit[17,4] := PLC_I_D17.4; //228
//	bInBit[17,5] := PLC_I_D17.5; //229
//	bInBit[17,6] := PLC_I_D17.6; //230
//	bInBit[17,7] := PLC_I_D17.7; //231
	
//	bInBit[18,0] := PLC_I_D18.0; //224
//	bInBit[18,1] := PLC_I_D18.1; //225
//	bInBit[18,2] := PLC_I_D18.2; //226
//	bInBit[18,3] := PLC_I_D18.3; //227
//	bInBit[18,4] := PLC_I_D18.4; //228
//	bInBit[18,5] := PLC_I_D18.5; //229
//	bInBit[18,6] := PLC_I_D18.6; //230
//	bInBit[18,7] := PLC_I_D18.7; //231
	
//	bInBit[19,0] := PLC_I_D19.0; //224
//	bInBit[19,1] := PLC_I_D19.1; //225
//	bInBit[19,2] := PLC_I_D19.2; //226
//	bInBit[19,3] := PLC_I_D19.3; //227
//	bInBit[19,4] := PLC_I_D19.4; //228
//	bInBit[19,5] := PLC_I_D19.5; //229
//	bInBit[19,6] := PLC_I_D19.6; //230
//	bInBit[19,7] := PLC_I_D19.7; //231
	
//	bInBit[20,0] := PLC_I_D20.0; //224
//	bInBit[20,1] := PLC_I_D20.1; //225
//	bInBit[20,2] := PLC_I_D20.2; //226
//	bInBit[20,3] := PLC_I_D20.3; //227
//	bInBit[20,4] := PLC_I_D20.4; //228
//	bInBit[20,5] := PLC_I_D20.5; //229
//	bInBit[20,6] := PLC_I_D20.6; //230
//	bInBit[20,7] := PLC_I_D20.7; //231
	
//	bInBit[21,0] := PLC_I_D21.0; //224
//	bInBit[21,1] := PLC_I_D21.1; //225
//	bInBit[21,2] := PLC_I_D21.2; //226
//	bInBit[21,3] := PLC_I_D21.3; //227
//	bInBit[21,4] := PLC_I_D21.4; //228
//	bInBit[21,5] := PLC_I_D21.5; //229
//	bInBit[21,6] := PLC_I_D21.6; //230
//	bInBit[21,7] := PLC_I_D21.7; //231
	
//	bInBit[22,0] := PLC_I_D22.0; //224
//	bInBit[22,1] := PLC_I_D22.1; //225
//	bInBit[22,2] := PLC_I_D22.2; //226
//	bInBit[22,3] := PLC_I_D22.3; //227
//	bInBit[22,4] := PLC_I_D22.4; //228
//	bInBit[22,5] := PLC_I_D22.5; //229
//	bInBit[22,6] := PLC_I_D22.6; //230
//	bInBit[22,7] := PLC_I_D22.7; //231
	
//	bInBit[23,0] := PLC_I_D23.0; //224
//	bInBit[23,1] := PLC_I_D23.1; //225
//	bInBit[23,2] := PLC_I_D23.2; //226
//	bInBit[23,3] := PLC_I_D23.3; //227
//	bInBit[23,4] := PLC_I_D23.4; //228
//	bInBit[23,5] := PLC_I_D23.5; //229
//	bInBit[23,6] := PLC_I_D23.6; //230
//	bInBit[23,7] := PLC_I_D23.7; //231
	
//	bInBit[24,0] := PLC_I_D24.0; //224
//	bInBit[24,1] := PLC_I_D24.1; //225
//	bInBit[24,2] := PLC_I_D24.2; //226
//	bInBit[24,3] := PLC_I_D24.3; //227
//	bInBit[24,4] := PLC_I_D24.4; //228
//	bInBit[24,5] := PLC_I_D24.5; //229
//	bInBit[24,6] := PLC_I_D24.6; //230
//	bInBit[24,7] := PLC_I_D24.7; //231
	
//	bInBit[25,0] := PLC_I_D25.0; //224
//	bInBit[25,1] := PLC_I_D25.1; //225
//	bInBit[25,2] := PLC_I_D25.2; //226
//	bInBit[25,3] := PLC_I_D25.3; //227
//	bInBit[25,4] := PLC_I_D25.4; //228
//	bInBit[25,5] := PLC_I_D25.5; //229
//	bInBit[25,6] := PLC_I_D25.6; //230
//	bInBit[25,7] := PLC_I_D25.7; //231
	
//	bInBit[26,0] := PLC_I_D26.0; //224
//	bInBit[26,1] := PLC_I_D26.1; //225
//	bInBit[26,2] := PLC_I_D26.2; //226
//	bInBit[26,3] := PLC_I_D26.3; //227
//	bInBit[26,4] := PLC_I_D26.4; //228
//	bInBit[26,5] := PLC_I_D26.5; //229
//	bInBit[26,6] := PLC_I_D26.6; //230
//	bInBit[26,7] := PLC_I_D26.7; //231
	
//	bInBit[27,0] := PLC_I_D27.0; //224
//	bInBit[27,1] := PLC_I_D27.1; //225
//	bInBit[27,2] := PLC_I_D27.2; //226
//	bInBit[27,3] := PLC_I_D27.3; //227
//	bInBit[27,4] := PLC_I_D27.4; //228
//	bInBit[27,5] := PLC_I_D27.5; //229
//	bInBit[27,6] := PLC_I_D27.6; //230
//	bInBit[27,7] := PLC_I_D27.7; //231
	
//	bInBit[28,0] := PLC_I_D28.0; //224
//	bInBit[28,1] := PLC_I_D28.1; //225
//	bInBit[28,2] := PLC_I_D28.2; //226
//	bInBit[28,3] := PLC_I_D28.3; //227
//	bInBit[28,4] := PLC_I_D28.4; //228
//	bInBit[28,5] := PLC_I_D28.5; //229
//	bInBit[28,6] := PLC_I_D28.6; //230
//	bInBit[28,7] := PLC_I_D28.7; //231
	
//	bInBit[29,0] := PLC_I_D29.0; //224
//	bInBit[29,1] := PLC_I_D29.1; //225
//	bInBit[29,2] := PLC_I_D29.2; //226
//	bInBit[29,3] := PLC_I_D29.3; //227
//	bInBit[29,4] := PLC_I_D29.4; //228
//	bInBit[29,5] := PLC_I_D29.5; //229
//	bInBit[29,6] := PLC_I_D29.6; //230
//	bInBit[29,7] := PLC_I_D29.7; //231
	
//	bInBit[30,0] := PLC_I_D30.0; //224
//	bInBit[30,1] := PLC_I_D30.1; //225
//	bInBit[30,2] := PLC_I_D30.2; //226
//	bInBit[30,3] := PLC_I_D30.3; //227
//	bInBit[30,4] := PLC_I_D30.4; //228
//	bInBit[30,5] := PLC_I_D30.5; //229
//	bInBit[30,6] := PLC_I_D30.6; //230
//	bInBit[30,7] := PLC_I_D30.7; //231
	
	//================================ Motion IO
	
//	IF NoMotion THEN
//		RETURN;
//	END_IF
	
//	PLC_O_D1.0 := bOutBit[1,0]; //200
//	PLC_O_D1.1 := bOutBit[1,1]; //201
//	PLC_O_D1.2 := bOutBit[1,2]; //202
//	PLC_O_D1.3 := bOutBit[1,3]; //203
//	PLC_O_D1.4 := bOutBit[1,4]; //204
//	PLC_O_D1.5 := bOutBit[1,5]; //205
//	PLC_O_D1.6 := bOutBit[1,6]; //206
//	PLC_O_D1.7 := bOutBit[1,7]; //207
	
//	PLC_O_D2.0 := bOutBit[2,0]; //208
//	PLC_O_D2.1 := bOutBit[2,1]; //209
//	PLC_O_D2.2 := bOutBit[2,2]; //210
//	PLC_O_D2.3 := bOutBit[2,3]; //211
//	PLC_O_D2.4 := bOutBit[2,4]; //212
//	PLC_O_D2.5 := bOutBit[2,5]; //213
//	PLC_O_D2.6 := bOutBit[2,6]; //214
//	PLC_O_D2.7 := bOutBit[2,7]; //215
	
//	PLC_O_D3.0 := bOutBit[3,0]; //216
//	PLC_O_D3.1 := bOutBit[3,1]; //217
//	PLC_O_D3.2 := bOutBit[3,2]; //218
//	PLC_O_D3.3 := bOutBit[3,3]; //219
//	PLC_O_D3.4 := bOutBit[3,4]; //220
//	PLC_O_D3.5 := bOutBit[3,5]; //221
//	PLC_O_D3.6 := bOutBit[3,6]; //222
//	PLC_O_D3.7 := bOutBit[3,7]; //223
	
//	bInBit[1,0] := PLC_I_D1.0; //200
//	bInBit[1,1] := PLC_I_D1.1; //201
//	bInBit[1,2] := PLC_I_D1.2; //202
//	bInBit[1,3] := PLC_I_D1.3; //203
//	bInBit[1,4] := PLC_I_D1.4; //204
//	bInBit[1,5] := PLC_I_D1.5; //205
//	bInBit[1,6] := PLC_I_D1.6; //206
//	bInBit[1,7] := PLC_I_D1.7; //207
	
//	bInBit[2,0] := PLC_I_D2.0; //208
//	bInBit[2,1] := PLC_I_D2.1; //209
//	bInBit[2,2] := PLC_I_D2.2; //210
//	bInBit[2,3] := PLC_I_D2.3; //211
//	bInBit[2,4] := PLC_I_D2.4; //212
//	bInBit[2,5] := PLC_I_D2.5; //213
//	bInBit[2,6] := PLC_I_D2.6; //214
//	bInBit[2,7] := PLC_I_D2.7; //215
	
//	bInBit[3,0] := PLC_I_D3.0; //216
//	bInBit[3,1] := PLC_I_D3.1; //217
//	bInBit[3,2] := PLC_I_D3.2; //218
//	bInBit[3,3] := PLC_I_D3.3; //219
//	bInBit[3,4] := PLC_I_D3.4; //220
//	bInBit[3,5] := PLC_I_D3.5; //221
//	bInBit[3,6] := PLC_I_D3.6; //222
//	bInBit[3,7] := PLC_I_D3.7; //223

END_PROGRAM

// ---- POUs/Kuka IO/KR2.TcPOU
// Programmed is linked to KR3
PROGRAM KR2

VAR_INPUT
	PLC_O_SYS 	AT %Q* : DWORD;
	PLC_O_PROG1 AT %Q* : DWORD;
	PLC_O_PROG2 AT %Q* : DWORD;
	
	PLC_I_SYS 	AT %I* : DWORD;
	PLC_I_PROG1 AT %I* : DWORD;
	PLC_I_PROG2 AT %I* : DWORD;
	PLC_I_AXIS 	AT %I* : ARRAY[1..6] OF DWORD;
	PLC_I_CURR	AT %I* : ARRAY[1..6] OF DWORD;
	PLC_I_TEMP	AT %I* : ARRAY[1..6] OF DWORD;

	KR2_Estop	: BOOL;
	Idle		: BOOL;
	NoMotion	: BOOL;
	
	index		: USINT;
	index1		: USINT;
	
	bOutBit 	: ARRAY [1..10,0..7] OF BOOL;
	bInBit  	: ARRAY [1..10,0..7] OF BOOL;
	
	dAxis		: ARRAY[1..6] OF DWORD;
	dCurr		: ARRAY[1..6] OF DWORD;
	dTemp		: ARRAY[1..6] OF DWORD;
END_VAR

VAR
	KROnline		: BOOL;
	KR_ProgReady	: BOOL;
END_VAR

	// =================================== If Soft EStop is pressed, turn off 1027 ~ 1034 
	IF KR2_Estop THEN		
		bOutBit[1,0]:=bOutBit[1,1]:=bOutBit[1,2]:=bOutBit[1,3]:=
		bOutBit[1,4]:=bOutBit[1,5]:=bOutBit[1,6]:=bOutBit[1,7]:=FALSE;
	END_IF

	// ============================================================================= Idle
	//Idle 	
	IF 	PLC_I_PROG1 = 1 AND PLC_I_PROG2 = 1 THEN 
			Idle := TRUE;
	ELSE
			Idle := FALSE;	
	END_IF
	
	
	// =========================================================================== Online 
	IF bInBit[1,0] OR bInBit[1,3] THEN
		KROnline := TRUE;
	ELSE
		KROnline := FALSE;
	END_IF

	// ===================================================================== Program Ready 
	IF bInBit[1,6] AND bInBit[2,4] THEN
		KR_ProgReady := TRUE;
	ELSIF GVL.KR3_bypass THEN
		KR_ProgReady := TRUE;
	ELSE
		KR_ProgReady := FALSE;
	END_IF
	
	// ======================================================================== System IO
	// Data In
	FOR index := 0 TO 31 BY 1 DO
		IF index < 8 THEN
			bInBit[1,index] := DWORD_TO_BOOL( SHR(PLC_I_SYS,index) AND 1);
		ELSIF index > 7 AND index < 16 THEN
			bInBit[2,index-8] := DWORD_TO_BOOL( SHR(PLC_I_SYS,index) AND 1);
		END_IF
	END_FOR
	
	// Data Out
	PLC_O_SYS.0 := bOutBit[1,0]; // 1027 move_enable
	PLC_O_SYS.1 := bOutBit[1,1]; // 1028 Drive_off
	PLC_O_SYS.2 := bOutBit[1,2]; // 1029 IO_Activate
	PLC_O_SYS.3 := bOutBit[1,3]; // 1030 Ext_Start
	PLC_O_SYS.4 := bOutBit[1,4]; // 1031 Conf_mess
	PLC_O_SYS.5 := bOutBit[1,5]; // 1032 
	PLC_O_SYS.6 := bOutBit[1,6]; // 1033 Drive_on
	PLC_O_SYS.7 := bOutBit[1,7]; // 1034 Pgno_Fbit
	PLC_O_SYS.8 := bOutBit[2,0]; // 1035 Pgno_Valid
	PLC_O_SYS.9 := bOutBit[2,1]; // 1036 Pgno_Parity

	// ===================================================================== Programme IO
	FOR index := 0 TO 31 BY 1 DO
		IF index < 8 THEN
			bInBit[3,index] := DWORD_TO_BOOL( SHR(PLC_I_PROG1,index) AND 1);
		ELSIF index > 7 AND index < 16 THEN
			bInBit[4,index-8] := DWORD_TO_BOOL( SHR(PLC_I_PROG1,index) AND 1);
		ELSIF index > 15 AND index < 24 THEN
			bInBit[5,index-16] := DWORD_TO_BOOL( SHR(PLC_I_PROG1,index) AND 1);
		ELSIF index > 23 THEN
			bInBit[6,index-24] := DWORD_TO_BOOL( SHR(PLC_I_PROG1,index) AND 1);
		END_IF
	END_FOR
	
	FOR index := 0 TO 31 BY 1 DO
		IF index < 8 THEN
			bInBit[7,index] := DWORD_TO_BOOL( SHR(PLC_I_PROG2,index) AND 1);
		ELSIF index > 7 AND index < 16 THEN
			bInBit[8,index-8] := DWORD_TO_BOOL( SHR(PLC_I_PROG2,index) AND 1);
//		ELSIF index > 15 AND index < 24 THEN
//			bInBit[9,index-16] := DWORD_TO_BOOL( SHR(PLC_I_PROG2,index) AND 1);
//		ELSIF index > 23 THEN
//			bInBit[10,index-24] := DWORD_TO_BOOL( SHR(PLC_I_PROG2,index) AND 1);
		END_IF
	END_FOR
	
	
	PLC_O_PROG1.0 := bOutBit[3,0]; // 200
	PLC_O_PROG1.1 := bOutBit[3,1]; // 201
	PLC_O_PROG1.2 := bOutBit[3,2]; // 202
	PLC_O_PROG1.3 := bOutBit[3,3]; // 203
	PLC_O_PROG1.4 := bOutBit[3,4]; // 204
	PLC_O_PROG1.5 := bOutBit[3,5]; // 205
	PLC_O_PROG1.6 := bOutBit[3,6]; // 206
	PLC_O_PROG1.7 := bOutBit[3,7]; // 207
	PLC_O_PROG1.8 := bOutBit[4,0]; // 208
	PLC_O_PROG1.9 := bOutBit[4,1]; // 209
	PLC_O_PROG1.10 := bOutBit[4,2]; // 210
	PLC_O_PROG1.11 := bOutBit[4,3]; // 211
	PLC_O_PROG1.12 := bOutBit[4,4]; // 212
	PLC_O_PROG1.13 := bOutBit[4,5]; // 213
	PLC_O_PROG1.14 := bOutBit[4,6]; // 214
	PLC_O_PROG1.15 := bOutBit[4,7]; // 215
	PLC_O_PROG1.16 := bOutBit[5,0]; // 216
	PLC_O_PROG1.17 := bOutBit[5,1]; // 217
	PLC_O_PROG1.18 := bOutBit[5,2]; // 218
	PLC_O_PROG1.19 := bOutBit[5,3]; // 219
	PLC_O_PROG1.20 := bOutBit[5,4]; // 220
	PLC_O_PROG1.21 := bOutBit[5,5]; // 221
	PLC_O_PROG1.22 := bOutBit[5,6]; // 222
	PLC_O_PROG1.23 := bOutBit[5,7]; // 223
	PLC_O_PROG1.24 := bOutBit[6,0]; // 224
	PLC_O_PROG1.25 := bOutBit[6,1]; // 225
	PLC_O_PROG1.26 := bOutBit[6,2]; // 226
	PLC_O_PROG1.27 := bOutBit[6,3]; // 227
	PLC_O_PROG1.28 := bOutBit[6,4]; // 228
	PLC_O_PROG1.29 := bOutBit[6,5]; // 229
	PLC_O_PROG1.30 := bOutBit[6,6]; // 230
	PLC_O_PROG1.31 := bOutBit[6,7]; // 231
	
	PLC_O_PROG2.0 := bOutBit[7,0]; // 232
	PLC_O_PROG2.1 := bOutBit[7,1]; // 233
	PLC_O_PROG2.2 := bOutBit[7,2]; // 234
	PLC_O_PROG2.3 := bOutBit[7,3]; // 235
	PLC_O_PROG2.4 := bOutBit[7,4]; // 236
	PLC_O_PROG2.5 := bOutBit[7,5]; // 237
	PLC_O_PROG2.6 := bOutBit[7,6]; // 238
	PLC_O_PROG2.7 := bOutBit[7,7]; // 239
	PLC_O_PROG2.8 := bOutBit[8,0]; // 240
	PLC_O_PROG2.9 := bOutBit[8,1]; // 241
	PLC_O_PROG2.10 := bOutBit[8,2]; // 242
	PLC_O_PROG2.11 := bOutBit[8,3]; // 243
	PLC_O_PROG2.12 := bOutBit[8,4]; // 244
	PLC_O_PROG2.13 := bOutBit[8,5]; // 245
	PLC_O_PROG2.14 := bOutBit[8,6]; // 246
	PLC_O_PROG2.15 := bOutBit[8,7]; // 247
	PLC_O_PROG2.16 := bOutBit[9,0]; // 248
	PLC_O_PROG2.17 := bOutBit[9,1]; // 249
	PLC_O_PROG2.18 := bOutBit[9,2]; // 250
	PLC_O_PROG2.19 := bOutBit[9,3]; // 251
	PLC_O_PROG2.20 := bOutBit[9,4]; // 252
	PLC_O_PROG2.21 := bOutBit[9,5]; // 253
	PLC_O_PROG2.22 := bOutBit[9,6]; // 254
	PLC_O_PROG2.23 := bOutBit[9,7]; // 255
	PLC_O_PROG2.24 := bOutBit[10,0]; // 256
	PLC_O_PROG2.25 := bOutBit[10,1]; // 257
	PLC_O_PROG2.26 := bOutBit[10,2]; // 258
	PLC_O_PROG2.27 := bOutBit[10,3]; // 259
	PLC_O_PROG2.28 := bOutBit[10,4]; // 260
	PLC_O_PROG2.29 := bOutBit[10,5]; // 261
	PLC_O_PROG2.30 := bOutBit[10,6]; // 262
	PLC_O_PROG2.31 := bOutBit[10,7]; // 263
	
	// ===================================================================== Robot Data
	FOR index1 := 1 TO 6 BY 1 DO
		FOR index := 0 TO 31 BY 1 DO
			dAxis[index1] := PLC_I_AXIS[index1];
			dCurr[index1] := PLC_I_CURR[index1];
			dTemp[index1] := PLC_I_TEMP[index1];
		END_FOR
	END_FOR
	
	
	
	
	
	
	
	
	
	
	
	
//	bInBit[2,0] := PLC_I_PROG1.0; // 200
//	bInBit[2,1] := PLC_I_PROG1.1; // 201
//	bInBit[2,2] := PLC_I_PROG1.2; // 202
//	bInBit[2,3] := PLC_I_PROG1.3; // 203
//	bInBit[2,4] := PLC_I_PROG1.4; // 204
//	bInBit[2,5] := PLC_I_PROG1.5; // 205
//	bInBit[2,6] := PLC_I_PROG1.6; // 206
//	bInBit[2,7] := PLC_I_PROG1.7; // 207
//	bInBit[2,8] := PLC_I_PROG1.8; // 208
//	bInBit[2,9] := PLC_I_PROG1.9; // 209
//	bInBit[2,10] := PLC_I_PROG1.10; // 210
//	bInBit[2,11] := PLC_I_PROG1.11; // 211
//	bInBit[2,12] := PLC_I_PROG1.12; // 212
//	bInBit[2,13] := PLC_I_PROG1.13; // 213
//	bInBit[2,14] := PLC_I_PROG1.14; // 214
//	bInBit[2,15] := PLC_I_PROG1.15; // 215
//	bInBit[2,16] := PLC_I_PROG1.16; // 216
//	bInBit[2,17] := PLC_I_PROG1.17; // 217
//	bInBit[2,18] := PLC_I_PROG1.18; // 218
//	bInBit[2,19] := PLC_I_PROG1.19; // 219
//	bInBit[2,20] := PLC_I_PROG1.20; // 220
//	bInBit[2,21] := PLC_I_PROG1.21; // 221
//	bInBit[2,22] := PLC_I_PROG1.22; // 222
//	bInBit[2,23] := PLC_I_PROG1.23; // 223
//	bInBit[2,24] := PLC_I_PROG1.24; // 224
//	bInBit[2,25] := PLC_I_PROG1.25; // 225
//	bInBit[2,26] := PLC_I_PROG1.26; // 226
//	bInBit[2,27] := PLC_I_PROG1.27; // 227
//	bInBit[2,28] := PLC_I_PROG1.28; // 228
//	bInBit[2,29] := PLC_I_PROG1.29; // 229
//	bInBit[2,30] := PLC_I_PROG1.30; // 230
//	bInBit[2,31] := PLC_I_PROG1.31; // 231
	
//	//================================ Function IO
	
//	PLC_O_D1.0 := bOutBit[1,0]; //1027 motion enable (on to start motor)
//	PLC_O_D1.1 := bOutBit[1,1]; //1028 Drives off (inverse) (on to start motor)
//	PLC_O_D1.2 := bOutBit[1,2]; //1029 Activate interface (on to start motor)
//	PLC_O_D1.3 := bOutBit[1,3]; //1030 Prog Start
//	PLC_O_D1.4 := bOutBit[1,4]; //1031 Acknowledge error msg
//	PLC_O_D1.5 := bOutBit[1,5]; //1032 Drives on
//	PLC_O_D1.6 := bOutBit[1,6]; //1033
//	PLC_O_D1.7 := bOutBit[1,7]; //1034
	
//	PLC_O_D2.0 := bOutBit[2,0]; //1035
//	PLC_O_D2.1 := bOutBit[2,1]; //1036
//	PLC_O_D2.2 := bOutBit[2,2]; //1037
//	PLC_O_D2.3 := bOutBit[2,3]; //1038
//	PLC_O_D2.4 := bOutBit[2,4]; //1039
//	PLC_O_D2.5 := bOutBit[2,5]; //1040
//	PLC_O_D2.6 := bOutBit[2,6]; //1041
//	PLC_O_D2.7 := bOutBit[2,7]; //1042
	
//	bInBit[1,0] := PLC_I_D1.0; //993
//	bInBit[1,1] := PLC_I_D1.1; //994
//	bInBit[1,2] := PLC_I_D1.2; //995
//	bInBit[1,3] := PLC_I_D1.3; //996
//	bInBit[1,4] := PLC_I_D1.4; //997
//	bInBit[1,5] := PLC_I_D1.5; //998
//	bInBit[1,6] := PLC_I_D1.6; //999
//	bInBit[1,7] := PLC_I_D1.7; //1000
	
//	bInBit[2,0] := PLC_I_D2.0; //1001
//	bInBit[2,1] := PLC_I_D2.1; //1002
//	bInBit[2,2] := PLC_I_D2.2; //1003
//	bInBit[2,3] := PLC_I_D2.3; //1004
//	bInBit[2,4] := PLC_I_D2.4; //1005
//	bInBit[2,5] := PLC_I_D2.5; //1006
//	bInBit[2,6] := PLC_I_D2.6; //1007
//	bInBit[2,7] := PLC_I_D2.7; //1008
	
//	//================================ Motion IO
	
//	IF NoMotion THEN
//		RETURN;
//	END_IF
	
//	PLC_O_D3.0 := bOutBit[3,0]; //200
//	PLC_O_D3.1 := bOutBit[3,1]; //201
//	PLC_O_D3.2 := bOutBit[3,2]; //202
//	PLC_O_D3.3 := bOutBit[3,3]; //203
//	PLC_O_D3.4 := bOutBit[3,4]; //204
//	PLC_O_D3.5 := bOutBit[3,5]; //205
//	PLC_O_D3.6 := bOutBit[3,6]; //206
//	PLC_O_D3.7 := bOutBit[3,7]; //207
	
//	PLC_O_D4.0 := bOutBit[4,0]; //208
//	PLC_O_D4.1 := bOutBit[4,1]; //209
//	PLC_O_D4.2 := bOutBit[4,2]; //210
//	PLC_O_D4.3 := bOutBit[4,3]; //211
//	PLC_O_D4.4 := bOutBit[4,4]; //212
//	PLC_O_D4.5 := bOutBit[4,5]; //213
//	PLC_O_D4.6 := bOutBit[4,6]; //214
//	PLC_O_D4.7 := bOutBit[4,7]; //215
	
//	PLC_O_D5.0 := bOutBit[5,0]; //216
//	PLC_O_D5.1 := bOutBit[5,1]; //217
//	PLC_O_D5.2 := bOutBit[5,2]; //218
//	PLC_O_D5.3 := bOutBit[5,3]; //219
//	PLC_O_D5.4 := bOutBit[5,4]; //220
//	PLC_O_D5.5 := bOutBit[5,5]; //221
//	PLC_O_D5.6 := bOutBit[5,6]; //222
//	PLC_O_D5.7 := bOutBit[5,7]; //223

//	PLC_O_D6.0 := bOutBit[6,0]; //224
//	PLC_O_D6.1 := bOutBit[6,1]; //225
//	PLC_O_D6.2 := bOutBit[6,2]; //226
//	PLC_O_D6.3 := bOutBit[6,3]; //227
//	PLC_O_D6.4 := bOutBit[6,4]; //228
//	PLC_O_D6.5 := bOutBit[6,5]; //229
//	PLC_O_D6.6 := bOutBit[6,6]; //230
//	PLC_O_D6.7 := bOutBit[6,7]; //231
	
//	PLC_O_D7.0 := bOutBit[7,0]; //216
//	PLC_O_D7.1 := bOutBit[7,1]; //217
//	PLC_O_D7.2 := bOutBit[7,2]; //218
//	PLC_O_D7.3 := bOutBit[7,3]; //219
//	PLC_O_D7.4 := bOutBit[7,4]; //220
//	PLC_O_D7.5 := bOutBit[7,5]; //221
//	PLC_O_D7.6 := bOutBit[7,6]; //222
//	PLC_O_D7.7 := bOutBit[7,7]; //223

//	PLC_O_D8.0 := bOutBit[8,0]; //224
//	PLC_O_D8.1 := bOutBit[8,1]; //225
//	PLC_O_D8.2 := bOutBit[8,2]; //226
//	PLC_O_D8.3 := bOutBit[8,3]; //227
//	PLC_O_D8.4 := bOutBit[8,4]; //228
//	PLC_O_D8.5 := bOutBit[8,5]; //229
//	PLC_O_D8.6 := bOutBit[8,6]; //230
//	PLC_O_D8.7 := bOutBit[8,7]; //231

//	bInBit[3,0] := PLC_I_D3.0; //200
//	bInBit[3,1] := PLC_I_D3.1; //201
//	bInBit[3,2] := PLC_I_D3.2; //202
//	bInBit[3,3] := PLC_I_D3.3; //203
//	bInBit[3,4] := PLC_I_D3.4; //204
//	bInBit[3,5] := PLC_I_D3.5; //205
//	bInBit[3,6] := PLC_I_D3.6; //206
//	bInBit[3,7] := PLC_I_D3.7; //207
	
//	bInBit[4,0] := PLC_I_D4.0; //208
//	bInBit[4,1] := PLC_I_D4.1; //209
//	bInBit[4,2] := PLC_I_D4.2; //210
//	bInBit[4,3] := PLC_I_D4.3; //211
//	bInBit[4,4] := PLC_I_D4.4; //212
//	bInBit[4,5] := PLC_I_D4.5; //213
//	bInBit[4,6] := PLC_I_D4.6; //214
//	bInBit[4,7] := PLC_I_D4.7; //215
	
//	bInBit[5,0] := PLC_I_D5.0; //216
//	bInBit[5,1] := PLC_I_D5.1; //217
//	bInBit[5,2] := PLC_I_D5.2; //218
//	bInBit[5,3] := PLC_I_D5.3; //219
//	bInBit[5,4] := PLC_I_D5.4; //220
//	bInBit[5,5] := PLC_I_D5.5; //221
//	bInBit[5,6] := PLC_I_D5.6; //222
//	bInBit[5,7] := PLC_I_D5.7; //223
	
//	bInBit[6,0] := PLC_I_D6.0; //224
//	bInBit[6,1] := PLC_I_D6.1; //225
//	bInBit[6,2] := PLC_I_D6.2; //226
//	bInBit[6,3] := PLC_I_D6.3; //227
//	bInBit[6,4] := PLC_I_D6.4; //228
//	bInBit[6,5] := PLC_I_D6.5; //229
//	bInBit[6,6] := PLC_I_D6.6; //230
//	bInBit[6,7] := PLC_I_D6.7; //231
	
//	bInBit[7,0] := PLC_I_D7.0; //224
//	bInBit[7,1] := PLC_I_D7.1; //225
//	bInBit[7,2] := PLC_I_D7.2; //226
//	bInBit[7,3] := PLC_I_D7.3; //227
//	bInBit[7,4] := PLC_I_D7.4; //228
//	bInBit[7,5] := PLC_I_D7.5; //229
//	bInBit[7,6] := PLC_I_D7.6; //230
//	bInBit[7,7] := PLC_I_D7.7; //231
	
//	bInBit[8,0] := PLC_I_D8.0; //224
//	bInBit[8,1] := PLC_I_D8.1; //225
//	bInBit[8,2] := PLC_I_D8.2; //226
//	bInBit[8,3] := PLC_I_D8.3; //227
//	bInBit[8,4] := PLC_I_D8.4; //228
//	bInBit[8,5] := PLC_I_D8.5; //229
//	bInBit[8,6] := PLC_I_D8.6; //230
//	bInBit[8,7] := PLC_I_D8.7; //231

END_PROGRAM

// ---- POUs/Kuka IO/KR3.TcPOU
PROGRAM KR3
VAR_INPUT
	
	PLC_O_SYS 	AT %Q* : DWORD;
	PLC_O_PROG1 AT %Q* : DWORD;
	
	PLC_I_SYS 	AT %I* : DWORD;
	PLC_I_PROG1 AT %I* : DWORD;
	PLC_I_AXIS 	AT %I* : ARRAY[1..6] OF DWORD;
	PLC_I_CURR	AT %I* : ARRAY[1..6] OF DWORD;
	PLC_I_TEMP	AT %I* : ARRAY[1..6] OF DWORD;
	
	KR3_Estop		: BOOL;
	Idle			: BOOL;
	NoMotion		: BOOL;
	
	bOutBit : ARRAY [1..3,0..7] OF BOOL;
	bInBit  : ARRAY [1..3,0..7] OF BOOL;
	
	index		: USINT;
	index1		: USINT;
	
	dAxis		: ARRAY[1..6] OF DWORD;
	dCurr		: ARRAY[1..6] OF DWORD;
	dTemp		: ARRAY[1..6] OF DWORD;
END_VAR

VAR
	KROnline: BOOL;
	KR_ProgReady: BOOL;
END_VAR

	//If Soft EStop is pressed, turn off 1027 ~ 1034
	IF KR3_Estop THEN		
		bOutBit[1,0]:=bOutBit[1,1]:=bOutBit[1,2]:=bOutBit[1,3]:=
		bOutBit[1,4]:=bOutBit[1,5]:=bOutBit[1,6]:=bOutBit[1,7]:=FALSE;
	END_IF

	//Idle 	
	IF 	PLC_I_PROG1 = 1 THEN 
			Idle := TRUE;
	ELSE
			Idle := FALSE;	
	END_IF
	
	//Online
	IF bInBit[1,0] OR bInBit[1,3] THEN
		KROnline := TRUE;
	ELSE
		KROnline := FALSE;
	END_IF

	//Program Ready
	IF bInBit[1,6] AND bInBit[2,4] THEN
		KR_ProgReady := TRUE;
	ELSIF GVL.KR2_bypass THEN
		KR_ProgReady := TRUE;
	ELSE
		KR_ProgReady := FALSE;
	END_IF
	
	// ======================================================================== System IO
	// Data In
	FOR index := 0 TO 31 BY 1 DO
		IF index < 8 THEN
			bInBit[1,index] := DWORD_TO_BOOL( SHR(PLC_I_SYS,index) AND 1);
		ELSIF index > 7 AND index < 16 THEN
			bInBit[2,index-8] := DWORD_TO_BOOL( SHR(PLC_I_SYS,index) AND 1);
		END_IF
	END_FOR
	
	// Data Out
	PLC_O_SYS.0 := bOutBit[1,0]; // 1027 move_enable
	PLC_O_SYS.1 := bOutBit[1,1]; // 1028 Drive_off
	PLC_O_SYS.2 := bOutBit[1,2]; // 1029 IO_Activate
	PLC_O_SYS.3 := bOutBit[1,3]; // 1030 Ext_Start
	PLC_O_SYS.4 := bOutBit[1,4]; // 1031 Conf_mess
	PLC_O_SYS.5 := bOutBit[1,5]; // 1032 Drive_on
	PLC_O_SYS.6 := bOutBit[1,6]; // 1033 Pgno_Fbit
	PLC_O_SYS.7 := bOutBit[1,7]; // 1034 Pgno_Valid
	PLC_O_SYS.8 := bOutBit[2,0]; // 1035 Pgno_Parity

	// ===================================================================== Programme IO
	FOR index := 0 TO 31 BY 1 DO
		IF index < 8 THEN
			bInBit[3,index] := DWORD_TO_BOOL( SHR(PLC_I_PROG1,index) AND 1);
		END_IF
	END_FOR
	
	PLC_O_PROG1.0 := bOutBit[3,0]; // 200
	PLC_O_PROG1.1 := bOutBit[3,1]; // 201
	PLC_O_PROG1.2 := bOutBit[3,2]; // 202
	PLC_O_PROG1.3 := bOutBit[3,3]; // 203
	PLC_O_PROG1.4 := bOutBit[3,4]; // 204
	PLC_O_PROG1.5 := bOutBit[3,5]; // 205
	PLC_O_PROG1.6 := bOutBit[3,6]; // 206
	PLC_O_PROG1.7 := bOutBit[3,7]; // 207
	
	// ===================================================================== Robot Data
	FOR index1 := 1 TO 6 BY 1 DO
		FOR index := 0 TO 31 BY 1 DO
			dAxis[index1] := PLC_I_AXIS[index1];
			dCurr[index1] := PLC_I_CURR[index1];
			dTemp[index1] := PLC_I_TEMP[index1];
		END_FOR
	END_FOR
	
	
	
	
	
	
//	//================================ Function IO
	
//	PLC_O_D1.0 := bOutBit[1,0]; //1027 motion enable (on to start motor)
//	PLC_O_D1.1 := bOutBit[1,1]; //1028 Drives off (inverse) (on to start motor)
//	PLC_O_D1.2 := bOutBit[1,2]; //1029 Activate interface (on to start motor)
//	PLC_O_D1.3 := bOutBit[1,3]; //1030 Prog Start
//	PLC_O_D1.4 := bOutBit[1,4]; //1031 Acknowledge error msg
//	PLC_O_D1.5 := bOutBit[1,5]; //1032 Drives on
//	PLC_O_D1.6 := bOutBit[1,6]; //1033
//	PLC_O_D1.7 := bOutBit[1,7]; //1034
	
//	PLC_O_D2.0 := bOutBit[2,0]; //1035
//	PLC_O_D2.1 := bOutBit[2,1]; //1036
//	PLC_O_D2.2 := bOutBit[2,2]; //1037
//	PLC_O_D2.3 := bOutBit[2,3]; //1038
//	PLC_O_D2.4 := bOutBit[2,4]; //1039
//	PLC_O_D2.5 := bOutBit[2,5]; //1040
//	PLC_O_D2.6 := bOutBit[2,6]; //1041
//	PLC_O_D2.7 := bOutBit[2,7]; //1042
	
//	bInBit[1,0] := PLC_I_D1.0; //993
//	bInBit[1,1] := PLC_I_D1.1; //994
//	bInBit[1,2] := PLC_I_D1.2; //995
//	bInBit[1,3] := PLC_I_D1.3; //996
//	bInBit[1,4] := PLC_I_D1.4; //997
//	bInBit[1,5] := PLC_I_D1.5; //998
//	bInBit[1,6] := PLC_I_D1.6; //999
//	bInBit[1,7] := PLC_I_D1.7; //1000
	
//	bInBit[2,0] := PLC_I_D2.0; //1001
//	bInBit[2,1] := PLC_I_D2.1; //1002
//	bInBit[2,2] := PLC_I_D2.2; //1003
//	bInBit[2,3] := PLC_I_D2.3; //1004
//	bInBit[2,4] := PLC_I_D2.4; //1005
//	bInBit[2,5] := PLC_I_D2.5; //1006
//	bInBit[2,6] := PLC_I_D2.6; //1007
//	bInBit[2,7] := PLC_I_D2.7; //1008
	
//	//================================ Motion IO
	
//	IF NoMotion THEN
//		RETURN;
//	END_IF
	
//	PLC_O_D3.0 := bOutBit[3,0]; //200
//	PLC_O_D3.1 := bOutBit[3,1]; //201
//	PLC_O_D3.2 := bOutBit[3,2]; //202
//	PLC_O_D3.3 := bOutBit[3,3]; //203
//	PLC_O_D3.4 := bOutBit[3,4]; //204
//	PLC_O_D3.5 := bOutBit[3,5]; //205
//	PLC_O_D3.6 := bOutBit[3,6]; //206
//	PLC_O_D3.7 := bOutBit[3,7]; //207

//	bInBit[3,0] := PLC_I_D3.0; //200
//	bInBit[3,1] := PLC_I_D3.1; //201
//	bInBit[3,2] := PLC_I_D3.2; //202
//	bInBit[3,3] := PLC_I_D3.3; //203
//	bInBit[3,4] := PLC_I_D3.4; //204
//	bInBit[3,5] := PLC_I_D3.5; //205
//	bInBit[3,6] := PLC_I_D3.6; //206
//	bInBit[3,7] := PLC_I_D3.7; //207

//	//If Soft EStop is pressed, turn off 1027, 1028, 1029, 1030, 1031
//	IF KR4_Estop THEN		
//		bOutBit[2,0]:=bOutBit[2,1]:=bOut
//	//If Soft EStop is pressed, turn off 1027, 1028, 1029, 1030, 1031
//	IF KR3_Estop THEN		
//		bOutBit[2,0]:=bOutBit[2,1]:=bOutBit[2,2]:=bOutBit[2,3]:=bOutBit[2,4]:=bOutBit[2,5]:=bOutBit[2,6]:=FALSE;
//	END_IF
	
//	//================================ Function IO

//	PLC_O_D2.0 := bOutBit[2,0]; //1027
//	PLC_O_D2.1 := bOutBit[2,1]; //1028
//	PLC_O_D2.2 := bOutBit[2,2]; //1029
//	PLC_O_D2.3 := bOutBit[2,3]; //1030
//	PLC_O_D2.4 := bOutBit[2,4]; //1031
//	PLC_O_D2.5 := bOutBit[2,5]; //1032
//	PLC_O_D2.6 := bOutBit[2,6]; //1033
//	PLC_O_D2.7 := bOutBit[2,7]; //1034
	
//	PLC_O_D3.0 := bOutBit[3,0]; //1035
//	PLC_O_D3.1 := bOutBit[3,1]; //1036
//	PLC_O_D3.2 := bOutBit[3,2]; //1037
//	PLC_O_D3.3 := bOutBit[3,3]; //1038
//	PLC_O_D3.4 := bOutBit[3,4]; //1039
//	PLC_O_D3.5 := bOutBit[3,5]; //1040
//	PLC_O_D3.6 := bOutBit[3,6]; //1041
//	PLC_O_D3.7 := bOutBit[3,7]; //1042
	
//	bInBit[2,0] := PLC_I_D2.0; //993
//	bInBit[2,1] := PLC_I_D2.1; //994
//	bInBit[2,2] := PLC_I_D2.2; //995
//	bInBit[2,3] := PLC_I_D2.3; //996
//	bInBit[2,4] := PLC_I_D2.4; //997
//	bInBit[2,5] := PLC_I_D2.5; //998
//	bInBit[2,6] := PLC_I_D2.6; //999
//	bInBit[2,7] := PLC_I_D2.7; //1000
	
//	bInBit[3,0] := PLC_I_D3.0; //1001
//	bInBit[3,1] := PLC_I_D3.1; //1002
//	bInBit[3,2] := PLC_I_D3.2; //1003
//	bInBit[3,3] := PLC_I_D3.3; //1004
//	bInBit[3,4] := PLC_I_D3.4; //1005
//	bInBit[3,5] := PLC_I_D3.5; //1006
//	bInBit[3,6] := PLC_I_D3.6; //1007
//	bInBit[3,7] := PLC_I_D3.7; //1008
	
//	//================================ Motion IO
	
//	IF NoMotion THEN
//		RETURN;
//	END_IF

//	PLC_O_D1.0 := bOutBit[1,0]; //300
//	PLC_O_D1.1 := bOutBit[1,1]; //301
//	PLC_O_D1.2 := bOutBit[1,2]; //302
//	PLC_O_D1.3 := bOutBit[1,3]; //303
//	PLC_O_D1.4 := bOutBit[1,4]; //304
//	PLC_O_D1.5 := bOutBit[1,5]; //305
//	PLC_O_D1.6 := bOutBit[1,6]; //306
//	PLC_O_D1.7 := bOutBit[1,7]; //307

//	bInBit[1,0] := PLC_I_D1.0; //300
//	bInBit[1,1] := PLC_I_D1.1; //301
//	bInBit[1,2] := PLC_I_D1.2; //302
//	bInBit[1,3] := PLC_I_D1.3; //303
//	bInBit[1,4] := PLC_I_D1.4; //304
//	bInBit[1,5] := PLC_I_D1.5; //305
//	bInBit[1,6] := PLC_I_D1.6; //306
//	bInBit[1,7] := PLC_I_D1.7; //307
	
//	IF PLC_I_D1 = 1 THEN
//		Idle := TRUE;
//	ELSE
//		Idle := FALSE;
//	END_IF

END_PROGRAM

// ---- POUs/Kuka IO/KR4.TcPOU
PROGRAM KR4
VAR_INPUT
	PLC_O_SYS 	AT %Q* : DWORD;
	PLC_O_PROG1 AT %Q* : DWORD;
	
	PLC_I_SYS 	AT %I* : DWORD;
	PLC_I_PROG1 AT %I* : DWORD;
	PLC_I_AXIS 	AT %I* : ARRAY[1..6] OF DWORD;
	PLC_I_CURR	AT %I* : ARRAY[1..6] OF DWORD;
	PLC_I_TEMP	AT %I* : ARRAY[1..6] OF DWORD;
	
	KR4_Estop		: BOOL;
	Idle			: BOOL;
	NoMotion		: BOOL;
	
	bOutBit : ARRAY [1..3,0..7] OF BOOL;
	bInBit  : ARRAY [1..3,0..7] OF BOOL;
	
	index		: USINT;
	index1		: USINT;
	
	dAxis		: ARRAY[1..6] OF DWORD;
	dCurr		: ARRAY[1..6] OF DWORD;
	dTemp		: ARRAY[1..6] OF DWORD;
END_VAR

VAR

	KROnline: BOOL;
	KR_ProgReady: BOOL;
END_VAR

	//If Soft EStop is pressed, turn off 1027 ~ 1034
	IF KR4_Estop THEN		
		bOutBit[1,0]:=bOutBit[1,1]:=bOutBit[1,2]:=bOutBit[1,3]:=
		bOutBit[1,4]:=bOutBit[1,5]:=bOutBit[1,6]:=bOutBit[1,7]:=FALSE;
	END_IF

	//Idle 	
	IF 	PLC_I_PROG1 = 1 THEN 
			Idle := TRUE;
	ELSE
			Idle := FALSE;	
	END_IF
	
	//Online
	IF bInBit[1,0] OR bInBit[1,3] THEN
		KROnline := TRUE;
	ELSE
		KROnline := FALSE;
	END_IF

	//Program Ready
	IF bInBit[1,6] AND bInBit[2,4] THEN
		KR_ProgReady := TRUE;
	ELSIF GVL.KR4_bypass THEN
		KR_ProgReady := TRUE;
	ELSE
		KR_ProgReady := FALSE;
	END_IF
	
	// ======================================================================== System IO
	// Data In
	FOR index := 0 TO 31 BY 1 DO
		IF index < 8 THEN
			bInBit[1,index] := DWORD_TO_BOOL( SHR(PLC_I_SYS,index) AND 1);
		ELSIF index > 7 AND index < 16 THEN
			bInBit[2,index-8] := DWORD_TO_BOOL( SHR(PLC_I_SYS,index) AND 1);
		END_IF
	END_FOR
	
	// Data Out
	PLC_O_SYS.0 := bOutBit[1,0]; // 1027 move_enable
	PLC_O_SYS.1 := bOutBit[1,1]; // 1028 Drive_off
	PLC_O_SYS.2 := bOutBit[1,2]; // 1029 IO_Activate
	PLC_O_SYS.3 := bOutBit[1,3]; // 1030 Ext_Start
	PLC_O_SYS.4 := bOutBit[1,4]; // 1031 Conf_mess
	PLC_O_SYS.5 := bOutBit[1,5]; // 1032 Drive_on
	PLC_O_SYS.6 := bOutBit[1,6]; // 1033 Pgno_Fbit
	PLC_O_SYS.7 := bOutBit[1,7]; // 1034 Pgno_Valid
	PLC_O_SYS.8 := bOutBit[2,0]; // 1035 Pgno_Parity

	// ===================================================================== Programme IO
	FOR index := 0 TO 31 BY 1 DO
		IF index < 8 THEN
			bInBit[3,index] := DWORD_TO_BOOL( SHR(PLC_I_PROG1,index) AND 1);
		END_IF
	END_FOR
	
	PLC_O_PROG1.0 := bOutBit[3,0]; // 200
	PLC_O_PROG1.1 := bOutBit[3,1]; // 201
	PLC_O_PROG1.2 := bOutBit[3,2]; // 202
	PLC_O_PROG1.3 := bOutBit[3,3]; // 203
	PLC_O_PROG1.4 := bOutBit[3,4]; // 204
	PLC_O_PROG1.5 := bOutBit[3,5]; // 205
	PLC_O_PROG1.6 := bOutBit[3,6]; // 206
	PLC_O_PROG1.7 := bOutBit[3,7]; // 207
	
	// ===================================================================== Robot Data
	FOR index1 := 1 TO 6 BY 1 DO
		FOR index := 0 TO 31 BY 1 DO
			dAxis[index1] := PLC_I_AXIS[index1];
			dCurr[index1] := PLC_I_CURR[index1];
			dTemp[index1] := PLC_I_TEMP[index1];
		END_FOR
	END_FOR
	
	
	
	
	
	
	
	
	
	
	
	
	
	
	
	
	
	
	
//	//================================ Function IO
	
//	PLC_O_D1.0 := bOutBit[1,0]; //1027 motion enable (on to start motor)
//	PLC_O_D1.1 := bOutBit[1,1]; //1028 Drives off (inverse) (on to start motor)
//	PLC_O_D1.2 := bOutBit[1,2]; //1029 Activate interface (on to start motor)
//	PLC_O_D1.3 := bOutBit[1,3]; //1030 Prog Start
//	PLC_O_D1.4 := bOutBit[1,4]; //1031 Acknowledge error msg
//	PLC_O_D1.5 := bOutBit[1,5]; //1032 Drives on
//	PLC_O_D1.6 := bOutBit[1,6]; //1033
//	PLC_O_D1.7 := bOutBit[1,7]; //1034
	
//	PLC_O_D2.0 := bOutBit[2,0]; //1035
//	PLC_O_D2.1 := bOutBit[2,1]; //1036
//	PLC_O_D2.2 := bOutBit[2,2]; //1037
//	PLC_O_D2.3 := bOutBit[2,3]; //1038
//	PLC_O_D2.4 := bOutBit[2,4]; //1039
//	PLC_O_D2.5 := bOutBit[2,5]; //1040
//	PLC_O_D2.6 := bOutBit[2,6]; //1041
//	PLC_O_D2.7 := bOutBit[2,7]; //1042
	
//	bInBit[1,0] := PLC_I_D1.0; //993
//	bInBit[1,1] := PLC_I_D1.1; //994
//	bInBit[1,2] := PLC_I_D1.2; //995
//	bInBit[1,3] := PLC_I_D1.3; //996
//	bInBit[1,4] := PLC_I_D1.4; //997
//	bInBit[1,5] := PLC_I_D1.5; //998
//	bInBit[1,6] := PLC_I_D1.6; //999
//	bInBit[1,7] := PLC_I_D1.7; //1000
	
//	bInBit[2,0] := PLC_I_D2.0; //1001
//	bInBit[2,1] := PLC_I_D2.1; //1002
//	bInBit[2,2] := PLC_I_D2.2; //1003
//	bInBit[2,3] := PLC_I_D2.3; //1004
//	bInBit[2,4] := PLC_I_D2.4; //1005
//	bInBit[2,5] := PLC_I_D2.5; //1006
//	bInBit[2,6] := PLC_I_D2.6; //1007
//	bInBit[2,7] := PLC_I_D2.7; //1008
	
//	//================================ Motion IO
	
//	IF NoMotion THEN
//		RETURN;
//	END_IF
	
//	PLC_O_D3.0 := bOutBit[3,0]; //200
//	PLC_O_D3.1 := bOutBit[3,1]; //201
//	PLC_O_D3.2 := bOutBit[3,2]; //202
//	PLC_O_D3.3 := bOutBit[3,3]; //203
//	PLC_O_D3.4 := bOutBit[3,4]; //204
//	PLC_O_D3.5 := bOutBit[3,5]; //205
//	PLC_O_D3.6 := bOutBit[3,6]; //206
//	PLC_O_D3.7 := bOutBit[3,7]; //207

//	bInBit[3,0] := PLC_I_D3.0; //200
//	bInBit[3,1] := PLC_I_D3.1; //201
//	bInBit[3,2] := PLC_I_D3.2; //202
//	bInBit[3,3] := PLC_I_D3.3; //203
//	bInBit[3,4] := PLC_I_D3.4; //204
//	bInBit[3,5] := PLC_I_D3.5; //205
//	bInBit[3,6] := PLC_I_D3.6; //206
//	bInBit[3,7] := PLC_I_D3.7; //207

	
